C05479=1171.912,88.058,-51.231,-179.130,6.211,148.864
C05480=1171.917,87.808,-51.214,-179.132,6.209,148.865
C05481=1171.922,87.559,-51.196,-179.135,6.209,148.865
C05482=1171.927,87.310,-51.178,-179.138,6.207,148.866
C05483=1171.932,87.061,-51.160,-179.140,6.206,148.866
C05484=1171.937,86.811,-51.142,-179.143,6.205,148.867
C05485=1171.942,86.562,-51.124,-179.145,6.204,148.867
C05486=1171.946,86.312,-51.108,-179.148,6.202,148.868
C05487=1171.951,86.063,-51.090,-179.150,6.202,148.868
C05488=1171.956,85.814,-51.072,-179.153,6.200,148.869
C05489=1171.961,85.564,-51.054,-179.156,6.198,148.869
C05490=1171.966,85.315,-51.037,-179.159,6.198,148.870
C05491=1171.971,85.067,-51.019,-179.162,6.196,148.871
C05492=1171.976,84.817,-51.002,-179.164,6.195,148.871
C05493=1171.981,84.568,-50.984,-179.167,6.194,148.872
C05494=1171.986,84.318,-50.967,-179.169,6.193,148.872
C05495=1171.991,84.069,-50.950,-179.172,6.191,148.872
C05496=1171.996,83.819,-50.932,-179.175,6.191,148.873
C05497=1172.001,83.570,-50.914,-179.177,6.189,148.874
C05498=1172.006,83.321,-50.896,-179.180,6.189,148.874
C05499=1172.010,83.071,-50.880,-179.183,6.187,148.875
C05500=1172.015,82.822,-50.862,-179.185,6.186,148.875
C05501=1172.020,82.572,-50.844,-179.188,6.185,148.876
C05502=1172.025,82.323,-50.826,-179.190,6.184,148.876
C05503=1172.030,82.074,-50.810,-179.193,6.182,148.877
C05504=1172.035,81.825,-50.792,-179.196,6.182,148.877
C05505=1172.040,81.575,-50.775,-179.199,6.180,148.878
C05506=1172.044,81.326,-50.757,-179.201,6.179,148.878
C05507=1172.050,81.077,-50.740,-179.204,6.178,148.879
C05508=1172.055,80.827,-50.723,-179.206,6.177,148.879
C05509=1172.060,80.559,-50.704,-179.209,6.175,148.880
C05510=1172.065,80.290,-50.686,-179.212,6.174,148.880
C05511=1172.071,80.022,-50.667,-179.215,6.173,148.881
C05512=1172.076,79.754,-50.648,-179.218,6.172,148.881
C05513=1172.080,79.504,-50.631,-179.221,6.171,148.882
C05514=1172.086,79.255,-50.614,-179.223,6.170,148.883
C05515=1172.090,79.005,-50.596,-179.226,6.168,148.883
C05516=1172.095,78.756,-50.579,-179.228,6.167,148.884
C05517=1172.101,78.507,-50.562,-179.231,6.166,148.884
C05518=1172.106,78.258,-50.544,-179.234,6.165,148.885
C05519=1172.110,78.008,-50.528,-179.236,6.163,148.885
C05520=1172.115,77.758,-50.510,-179.239,6.163,148.886
C05521=1172.120,77.510,-50.493,-179.242,6.161,148.886
C05522=1172.125,77.260,-50.476,-179.244,6.161,148.887
C05523=1172.130,77.011,-50.459,-179.247,6.159,148.887
C05524=1172.135,76.762,-50.441,-179.250,6.159,148.888
C05525=1172.140,76.512,-50.424,-179.252,6.157,148.888
C05526=1172.144,76.262,-50.408,-179.255,6.156,148.889
C05527=1172.150,76.013,-50.390,-179.258,6.155,148.889
C05528=1172.154,75.765,-50.373,-179.260,6.154,148.890
C05529=1172.160,75.515,-50.356,-179.263,6.153,148.891
C05530=1172.164,75.265,-50.339,-179.265,6.152,148.891
C05531=1172.169,75.015,-50.322,-179.268,6.151,148.892
C05532=1172.174,74.766,-50.305,-179.271,6.149,148.892
C05533=1172.179,74.517,-50.288,-179.273,6.149,148.893
C05534=1172.184,74.268,-50.271,-179.276,6.147,148.893
C05535=1172.189,74.018,-50.254,-179.279,6.147,148.894
C05536=1172.193,73.769,-50.237,-179.281,6.145,148.894
C05537=1172.199,73.519,-50.220,-179.283,6.144,148.895
C05538=1172.204,73.270,-50.204,-179.287,6.143,148.895
C05539=1172.209,73.021,-50.186,-179.289,6.142,148.896
C05540=1172.213,72.771,-50.169,-179.292,6.140,148.896
C05541=1172.218,72.522,-50.152,-179.294,6.140,148.897
C05542=1172.223,72.273,-50.135,-179.297,6.139,148.898
C05543=1172.229,72.023,-50.118,-179.300,6.137,148.898
C05544=1172.233,71.774,-50.101,-179.302,6.137,148.899
C05545=1172.238,71.524,-50.085,-179.305,6.135,148.899
C05546=1172.243,71.275,-50.068,-179.308,6.135,148.900
C05547=1172.248,71.026,-50.051,-179.310,6.133,148.900
C05548=1172.253,70.776,-50.034,-179.313,6.132,148.901
C05549=1172.258,70.527,-50.018,-179.316,6.131,148.901
C05550=1172.263,70.277,-50.001,-179.318,6.130,148.902
C05551=1172.268,70.028,-49.984,-179.320,6.129,148.902
C05552=1172.272,69.778,-49.967,-179.323,6.128,148.903
C05553=1172.278,69.530,-49.949,-179.326,6.127,148.903
C05554=1172.283,69.280,-49.933,-179.329,6.125,148.904
C05555=1172.287,69.030,-49.917,-179.331,6.125,148.904
C05556=1172.293,68.781,-49.900,-179.334,6.123,148.905
C05557=1172.298,68.532,-49.883,-179.337,6.123,148.906
C05558=1172.302,68.282,-49.867,-179.339,6.122,148.906
C05559=1172.308,68.033,-49.850,-179.342,6.120,148.907
C05560=1172.312,67.784,-49.833,-179.344,6.120,148.907
C05561=1172.317,67.534,-49.816,-179.347,6.118,148.908
C05562=1172.323,67.285,-49.799,-179.349,6.117,148.908
C05563=1172.327,67.035,-49.783,-179.353,6.116,148.909
C05564=1172.332,66.786,-49.766,-179.355,6.115,148.909
C05565=1172.337,66.537,-49.749,-179.357,6.115,148.910
C05566=1172.342,66.287,-49.733,-179.360,6.113,148.910
C05567=1172.346,66.038,-49.716,-179.363,6.112,148.911
C05568=1172.352,65.789,-49.700,-179.365,6.111,148.911
C05569=1172.357,65.539,-49.683,-179.368,6.110,148.912
C05570=1172.362,65.290,-49.667,-179.370,6.109,148.913
C05571=1172.367,65.040,-49.650,-179.373,6.108,148.913
C05572=1172.371,64.791,-49.633,-179.376,6.107,148.914
C05573=1172.377,64.542,-49.616,-179.379,6.106,148.914
C05574=1172.382,64.292,-49.600,-179.381,6.105,148.915
C05575=1172.386,64.042,-49.584,-179.384,6.104,148.915
C05576=1172.391,63.793,-49.568,-179.386,6.103,148.916
C05577=1172.396,63.544,-49.550,-179.389,6.102,148.916
C05578=1172.401,63.295,-49.534,-179.392,6.101,148.917
C05579=1172.406,63.045,-49.518,-179.394,6.100,148.918
C05580=1172.411,62.796,-49.502,-179.397,6.099,148.918
C05581=1172.416,62.547,-49.485,-179.400,6.098,148.919
C05582=1172.421,62.296,-49.468,-179.402,6.097,148.919
C05583=1172.426,62.047,-49.452,-179.405,6.096,148.920
C05584=1172.431,61.798,-49.436,-179.407,6.095,148.920
C05585=1172.436,61.549,-49.419,-179.410,6.094,148.921
C05586=1172.441,61.299,-49.403,-179.413,6.093,148.921
C05587=1172.446,61.050,-49.387,-179.415,6.092,148.922
C05588=1172.450,60.801,-49.370,-179.417,6.091,148.922
C05589=1172.456,60.550,-49.354,-179.421,6.090,148.923
C05590=1172.461,60.302,-49.337,-179.423,6.089,148.924
C05591=1172.465,60.052,-49.321,-179.426,6.088,148.924
C05592=1172.471,59.803,-49.305,-179.428,6.087,148.925
C05593=1172.475,59.553,-49.289,-179.431,6.086,148.925
C05594=1172.481,59.304,-49.273,-179.434,6.085,148.926
C05595=1172.485,59.054,-49.256,-179.436,6.084,148.926
C05596=1172.490,58.805,-49.240,-179.438,6.083,148.927
C05597=1172.495,58.555,-49.224,-179.442,6.082,148.927
C05598=1172.501,58.306,-49.207,-179.444,6.081,148.928
C05599=1172.506,58.056,-49.191,-179.447,6.080,148.929
C05600=1172.511,57.807,-49.175,-179.449,6.079,148.929
C05601=1172.515,57.558,-49.158,-179.452,6.078,148.930
C05602=1172.521,57.308,-49.143,-179.454,6.077,148.930
C05603=1172.525,57.059,-49.126,-179.457,6.076,148.931
C05604=1172.530,56.810,-49.110,-179.459,6.075,148.931
C05605=1172.535,56.560,-49.094,-179.462,6.074,148.932
C05606=1172.540,56.311,-49.078,-179.465,6.073,148.932
C05607=1172.545,56.061,-49.061,-179.467,6.073,148.933
C05608=1172.550,55.812,-49.046,-179.470,6.071,148.934
C05609=1172.555,55.563,-49.030,-179.473,6.070,148.934
C05610=1172.560,55.313,-49.014,-179.475,6.070,148.935
C05611=1172.565,55.064,-48.998,-179.478,6.068,148.935
C05612=1172.570,54.814,-48.981,-179.481,6.068,148.936
C05613=1172.575,54.546,-48.964,-179.483,6.066,148.936
C05614=1172.581,54.277,-48.947,-179.486,6.065,148.937
C05615=1172.586,54.008,-48.930,-179.489,6.064,148.938
C05616=1172.591,53.740,-48.912,-179.492,6.064,148.938
C05617=1172.597,53.491,-48.897,-179.494,6.063,148.939
C05618=1172.601,53.241,-48.881,-179.497,6.061,148.939
C05619=1172.606,52.992,-48.864,-179.499,6.061,148.940
C05620=1172.612,52.742,-48.849,-179.502,6.060,148.941
C05621=1172.616,52.493,-48.832,-179.505,6.058,148.941
C05622=1172.622,52.243,-48.816,-179.507,6.058,148.942
C05623=1172.626,51.993,-48.800,-179.510,6.057,148.942
C05624=1172.632,51.745,-48.784,-179.513,6.056,148.943
C05625=1172.637,51.495,-48.769,-179.515,6.055,148.943
C05626=1172.641,51.245,-48.753,-179.518,6.054,148.944
C05627=1172.646,50.997,-48.737,-179.520,6.053,148.944
C05628=1172.651,50.747,-48.721,-179.523,6.052,148.945
C05629=1172.656,50.497,-48.705,-179.526,6.052,148.946
C05630=1172.662,50.248,-48.690,-179.528,6.050,148.946
C05631=1172.666,49.998,-48.673,-179.531,6.049,148.947
C05632=1172.672,49.749,-48.658,-179.533,6.049,148.947
C05633=1172.677,49.499,-48.642,-179.536,6.047,148.948
C05634=1172.681,49.250,-48.627,-179.538,6.046,148.948
C05635=1172.686,49.001,-48.610,-179.541,6.046,148.949
C05636=1172.691,48.751,-48.594,-179.544,6.044,148.949
C05637=1172.696,48.501,-48.579,-179.547,6.044,148.950
C05638=1172.702,48.252,-48.563,-179.549,6.043,148.950
C05639=1172.705,48.003,-48.547,-179.551,6.042,148.951
C05640=1172.711,47.753,-48.532,-179.555,6.041,148.952
C05641=1172.716,47.504,-48.516,-179.557,6.040,148.952
C05642=1172.721,47.255,-48.500,-179.559,6.040,148.953
C05643=1172.726,47.004,-48.484,-179.562,6.038,148.953
C05644=1172.731,46.755,-48.469,-179.565,6.038,148.954
C05645=1172.736,46.507,-48.453,-179.567,6.037,148.954
C05646=1172.741,46.256,-48.437,-179.569,6.036,148.955
C05647=1172.746,46.007,-48.422,-179.572,6.034,148.956
C05648=1172.752,45.758,-48.406,-179.575,6.034,148.956
C05649=1172.756,45.508,-48.391,-179.578,6.033,148.957
C05650=1172.761,45.258,-48.375,-179.580,6.032,148.957
C05651=1172.766,45.009,-48.359,-179.583,6.031,148.958
C05652=1172.771,44.760,-48.344,-179.585,6.030,148.959
C05653=1172.776,44.510,-48.328,-179.588,6.030,148.959
C05654=1172.781,44.260,-48.313,-179.590,6.028,148.960
C05655=1172.787,44.011,-48.297,-179.593,6.028,148.960
C05656=1172.791,43.761,-48.282,-179.595,6.027,148.961
C05657=1172.796,43.513,-48.266,-179.598,6.026,148.961
C05658=1172.801,43.263,-48.250,-179.601,6.025,148.962
C05659=1172.806,43.014,-48.235,-179.603,6.024,148.963
C05660=1172.811,42.765,-48.219,-179.606,6.024,148.963
C05661=1172.816,42.515,-48.204,-179.609,6.022,148.964
C05662=1172.821,42.265,-48.189,-179.611,6.022,148.964
C05663=1172.826,42.016,-48.173,-179.613,6.021,148.965
C05664=1172.832,41.766,-48.158,-179.616,6.020,148.965
C05665=1172.836,41.516,-48.143,-179.619,6.019,148.966
C05666=1172.841,41.267,-48.127,-179.621,6.018,148.967
C05667=1172.846,41.017,-48.112,-179.624,6.018,148.967
C05668=1172.851,40.768,-48.097,-179.626,6.017,148.968
C05669=1172.857,40.519,-48.081,-179.629,6.015,148.968
C05670=1172.861,40.269,-48.065,-179.632,6.014,148.969
C05671=1172.866,40.020,-48.050,-179.634,6.014,148.969
C05672=1172.871,39.770,-48.034,-179.637,6.014,148.970
C05673=1172.876,39.521,-48.019,-179.640,6.012,148.971
C05674=1172.881,39.272,-48.004,-179.642,6.011,148.971
C05675=1172.886,39.022,-47.988,-179.644,6.010,148.972
C05676=1172.891,38.772,-47.974,-179.647,6.010,148.972
C05677=1172.897,38.523,-47.958,-179.650,6.008,148.973
C05678=1172.901,38.274,-47.943,-179.653,6.008,148.973
C05679=1172.907,38.024,-47.927,-179.655,6.007,148.974
C05680=1172.911,37.775,-47.912,-179.657,6.006,148.975
C05681=1172.916,37.525,-47.896,-179.661,6.005,148.975
C05682=1172.922,37.275,-47.882,-179.663,6.004,148.976
C05683=1172.926,37.026,-47.867,-179.665,6.004,148.976
C05684=1172.932,36.776,-47.851,-179.668,6.003,148.977
C05685=1172.936,36.527,-47.836,-179.670,6.002,148.978
C05686=1172.942,36.278,-47.820,-179.673,6.001,148.978
C05687=1172.947,36.028,-47.806,-179.676,6.000,148.979
C05688=1172.952,35.779,-47.791,-179.678,6.000,148.979
C05689=1172.956,35.529,-47.775,-179.680,5.999,148.980
C05690=1172.962,35.280,-47.760,-179.684,5.998,148.980
C05691=1172.966,35.030,-47.745,-179.686,5.997,148.981
C05692=1172.972,34.780,-47.730,-179.688,5.996,148.982
C05693=1172.977,34.531,-47.715,-179.691,5.996,148.982
C05694=1172.982,34.281,-47.700,-179.693,5.995,148.983
C05695=1172.987,34.032,-47.685,-179.696,5.994,148.983
C05696=1172.992,33.783,-47.669,-179.699,5.993,148.984
C05697=1172.997,33.533,-47.655,-179.701,5.992,148.984
C05698=1173.001,33.283,-47.640,-179.704,5.992,148.985
C05699=1173.007,33.034,-47.624,-179.707,5.990,148.986
C05700=1173.012,32.784,-47.610,-179.709,5.990,148.986
C05701=1173.017,32.535,-47.594,-179.711,5.989,148.987
C05702=1173.022,32.286,-47.579,-179.714,5.988,148.987
C05703=1173.027,32.036,-47.564,-179.717,5.988,148.988
C05704=1173.032,31.787,-47.549,-179.719,5.986,148.989
C05705=1173.037,31.537,-47.535,-179.722,5.986,148.989
C05706=1173.042,31.288,-47.520,-179.724,5.985,148.990
C05707=1173.047,31.038,-47.505,-179.727,5.984,148.990
C05708=1173.053,30.788,-47.490,-179.730,5.984,148.991
C05709=1173.057,30.539,-47.475,-179.732,5.982,148.991
C05710=1173.062,30.290,-47.460,-179.735,5.982,148.992
C05711=1173.068,30.040,-47.445,-179.737,5.981,148.993
C05712=1173.073,29.791,-47.431,-179.740,5.980,148.993
C05713=1173.077,29.541,-47.416,-179.742,5.980,148.994
C05714=1173.083,29.292,-47.400,-179.745,5.979,148.994
C05715=1173.088,29.042,-47.386,-179.748,5.978,148.995
C05716=1173.092,28.793,-47.371,-179.750,5.977,148.996
C05717=1173.098,28.524,-47.354,-179.753,5.976,148.996
C05718=1173.103,28.255,-47.339,-179.756,5.975,148.997
C05719=1173.109,27.986,-47.322,-179.758,5.975,148.998
C05720=1173.114,27.717,-47.307,-179.761,5.974,148.998
C05721=1173.119,27.468,-47.292,-179.763,5.973,148.999
C05722=1173.125,27.218,-47.277,-179.767,5.972,148.999
C05723=1173.130,26.969,-47.263,-179.769,5.971,149.000
C05724=1173.134,26.720,-47.248,-179.771,5.971,149.001
C05725=1173.139,26.470,-47.233,-179.774,5.970,149.001
C05726=1173.145,26.220,-47.218,-179.776,5.969,149.002
C05727=1173.149,25.971,-47.203,-179.779,5.969,149.002
C05728=1173.154,25.721,-47.189,-179.782,5.967,149.003
C05729=1173.159,25.472,-47.174,-179.784,5.967,149.003
C05730=1173.165,25.222,-47.159,-179.787,5.966,149.004
C05731=1173.170,24.972,-47.145,-179.789,5.965,149.005
C05732=1173.174,24.723,-47.130,-179.792,5.965,149.005
C05733=1173.179,24.473,-47.116,-179.794,5.964,149.006
C05734=1173.185,24.223,-47.101,-179.797,5.963,149.006
C05735=1173.190,23.974,-47.086,-179.800,5.962,149.007
C05736=1173.195,23.725,-47.072,-179.802,5.961,149.008
C05737=1173.200,23.476,-47.058,-179.804,5.961,149.008
C05738=1173.205,23.226,-47.043,-179.807,5.960,149.009
C05739=1173.211,22.976,-47.028,-179.809,5.960,149.009
C05740=1173.215,22.727,-47.013,-179.812,5.959,149.010
C05741=1173.220,22.478,-46.999,-179.815,5.957,149.010
C05742=1173.225,22.228,-46.984,-179.817,5.957,149.011
C05743=1173.230,21.978,-46.970,-179.820,5.956,149.012
C05744=1173.235,21.728,-46.956,-179.822,5.956,149.012
C05745=1173.240,21.479,-46.940,-179.825,5.955,149.013
C05746=1173.245,21.229,-46.926,-179.827,5.954,149.013
C05747=1173.251,20.980,-46.912,-179.830,5.954,149.014
C05748=1173.256,20.731,-46.898,-179.833,5.953,149.015
C05749=1173.260,20.482,-46.883,-179.835,5.952,149.015
C05750=1173.265,20.232,-46.868,-179.838,5.951,149.016
C05751=1173.270,19.982,-46.854,-179.840,5.950,149.016
C05752=1173.276,19.732,-46.839,-179.842,5.950,149.017
C05753=1173.281,19.482,-46.825,-179.845,5.949,149.018
C05754=1173.286,19.233,-46.811,-179.847,5.949,149.018
C05755=1173.291,18.984,-46.796,-179.851,5.947,149.019
C05756=1173.296,18.735,-46.782,-179.853,5.946,149.019
C05757=1173.301,18.485,-46.767,-179.855,5.946,149.020
C05758=1173.306,18.235,-46.753,-179.858,5.945,149.021
C05759=1173.311,17.985,-46.739,-179.860,5.945,149.021
C05760=1173.316,17.736,-46.725,-179.863,5.944,149.022
C05761=1173.322,17.487,-46.711,-179.865,5.944,149.023
C05762=1173.326,17.238,-46.696,-179.868,5.943,149.023
C05763=1173.331,16.988,-46.681,-179.870,5.942,149.024
C05764=1173.336,16.738,-46.667,-179.873,5.941,149.024
C05765=1173.341,16.489,-46.653,-179.876,5.940,149.025
C05766=1173.347,16.240,-46.639,-179.878,5.940,149.025
C05767=1173.352,15.990,-46.625,-179.880,5.939,149.026
C05768=1173.357,15.740,-46.610,-179.883,5.938,149.027
C05769=1173.361,15.490,-46.596,-179.886,5.938,149.027
C05770=1173.366,15.241,-46.582,-179.888,5.937,149.028
C05771=1173.372,14.992,-46.568,-179.891,5.937,149.028
C05772=1173.377,14.742,-46.554,-179.893,5.936,149.029
C05773=1173.382,14.492,-46.539,-179.896,5.934,149.030
C05774=1173.387,14.243,-46.525,-179.899,5.934,149.030
C05775=1173.392,13.993,-46.511,-179.901,5.933,149.031
C05776=1173.397,13.744,-46.497,-179.903,5.933,149.031
C05777=1173.402,13.494,-46.483,-179.906,5.932,149.032
C05778=1173.407,13.244,-46.468,-179.908,5.931,149.033
C05779=1173.412,12.995,-46.454,-179.911,5.931,149.033
C05780=1173.418,12.746,-46.440,-179.913,5.930,149.034
C05781=1173.423,12.496,-46.426,-179.916,5.930,149.034
C05782=1173.428,12.246,-46.412,-179.918,5.929,149.035
C05783=1173.433,11.997,-46.397,-179.921,5.928,149.035
C05784=1173.438,11.748,-46.383,-179.924,5.927,149.036
C05785=1173.443,11.498,-46.369,-179.926,5.927,149.037
C05786=1173.448,11.247,-46.356,-179.929,5.926,149.037
C05787=1173.453,10.998,-46.341,-179.931,5.925,149.038
C05788=1173.458,10.749,-46.328,-179.933,5.924,149.038
C05789=1173.463,10.499,-46.314,-179.936,5.924,149.039
C05790=1173.468,10.250,-46.299,-179.939,5.923,149.040
C05791=1173.474,10.001,-46.286,-179.941,5.923,149.040
C05792=1173.479,9.751,-46.271,-179.944,5.922,149.041
C05793=1173.484,9.501,-46.257,-179.946,5.922,149.042
C05794=1173.489,9.252,-46.244,-179.948,5.921,149.042
C05795=1173.494,9.002,-46.230,-179.951,5.920,149.043
C05796=1173.499,8.752,-46.216,-179.954,5.920,149.043
C05797=1173.504,8.503,-46.202,-179.956,5.918,149.044
C05798=1173.509,8.254,-46.188,-179.959,5.918,149.045
C05799=1173.514,8.003,-46.174,-179.961,5.917,149.045
C05800=1173.519,7.754,-46.160,-179.964,5.916,149.046
C05801=1173.525,7.505,-46.146,-179.967,5.916,149.046
C05802=1173.529,7.255,-46.132,-179.969,5.915,149.047
C05803=1173.534,7.005,-46.119,-179.971,5.915,149.048
C05804=1173.540,6.756,-46.105,-179.974,5.914,149.048
C05805=1173.545,6.506,-46.090,-179.976,5.913,149.049
C05806=1173.550,6.257,-46.076,-179.979,5.913,149.049
C05807=1173.555,6.007,-46.064,-179.982,5.912,149.050
C05808=1173.560,5.758,-46.049,-179.984,5.912,149.051
C05809=1173.565,5.509,-46.035,-179.986,5.911,149.051
C05810=1173.570,5.259,-46.021,-179.989,5.910,149.052
C05811=1173.575,5.009,-46.008,-179.991,5.910,149.052
C05812=1173.581,4.760,-45.994,-179.994,5.909,149.053
C05813=1173.585,4.510,-45.980,-179.996,5.908,149.054
C05814=1173.591,4.260,-45.966,-179.999,5.908,149.054
C05815=1173.596,4.011,-45.953,179.999,5.908,149.055
C05816=1173.601,3.761,-45.939,179.996,5.906,149.055
C05817=1173.606,3.512,-45.926,179.993,5.905,149.056
C05818=1173.611,3.262,-45.912,179.991,5.905,149.057
C05819=1173.616,3.012,-45.898,179.988,5.904,149.057
C05820=1173.621,2.763,-45.884,179.986,5.904,149.058
C05821=1173.627,2.494,-45.869,179.983,5.903,149.059
C05822=1173.632,2.224,-45.854,179.981,5.903,149.059
C05823=1173.637,1.955,-45.840,179.978,5.902,149.060
C05824=1173.643,1.686,-45.825,179.976,5.901,149.060
C05825=1173.648,1.436,-45.812,179.973,5.901,149.061
C05826=1173.654,1.187,-45.798,179.970,5.899,149.062
C05827=1173.658,0.937,-45.785,179.968,5.899,149.062
C05828=1173.663,0.687,-45.771,179.965,5.898,149.063
C05829=1173.669,0.438,-45.758,179.963,5.898,149.063
C05830=1173.673,0.188,-45.744,179.960,5.897,149.064
C05831=1173.679,-0.061,-45.731,179.957,5.897,149.065
C05832=1173.683,-0.311,-45.717,179.955,5.896,149.065
C05833=1173.689,-0.560,-45.704,179.953,5.895,149.066
C05834=1173.694,-0.810,-45.690,179.950,5.895,149.067
C05835=1173.699,-1.059,-45.677,179.948,5.894,149.067
C05836=1173.704,-1.309,-45.663,179.945,5.894,149.068
C05837=1173.710,-1.559,-45.649,179.943,5.893,149.069
C05838=1173.714,-1.808,-45.636,179.940,5.892,149.069
C05839=1173.720,-2.058,-45.623,179.938,5.892,149.070
C05840=1173.724,-2.307,-45.609,179.936,5.891,149.070
C05841=1173.730,-2.557,-45.596,179.933,5.891,149.071
C05842=1173.735,-2.807,-45.581,179.930,5.890,149.071
C05843=1173.740,-3.056,-45.569,179.928,5.889,149.072
C05844=1173.746,-3.306,-45.555,179.925,5.889,149.073
C05845=1173.751,-3.555,-45.542,179.923,5.888,149.073
C05846=1173.756,-3.805,-45.528,179.921,5.887,149.074
C05847=1173.761,-4.054,-45.515,179.918,5.887,149.074
C05848=1173.766,-4.304,-45.501,179.915,5.887,149.075
C05849=1173.771,-4.554,-45.489,179.913,5.886,149.076
C05850=1173.776,-4.803,-45.475,179.910,5.885,149.076
C05851=1173.781,-5.053,-45.462,179.908,5.885,149.077
C05852=1173.786,-5.303,-45.448,179.906,5.884,149.077
C05853=1173.791,-5.552,-45.435,179.903,5.884,149.078
C05854=1173.796,-5.802,-45.422,179.900,5.883,149.079
C05855=1173.802,-6.051,-45.409,179.898,5.882,149.079
C05856=1173.806,-6.301,-45.395,179.895,5.882,149.080
C05857=1173.812,-6.550,-45.382,179.893,5.881,149.080
C05858=1173.817,-6.801,-45.369,179.891,5.880,149.081
C05859=1173.822,-7.049,-45.355,179.888,5.880,149.082
C05860=1173.828,-7.299,-45.342,179.886,5.879,149.082
C05861=1173.832,-7.549,-45.329,179.883,5.879,149.083
C05862=1173.838,-7.799,-45.316,179.880,5.878,149.084
C05863=1173.842,-8.048,-45.302,179.878,5.877,149.084
C05864=1173.848,-8.298,-45.289,179.876,5.877,149.085
C05865=1173.853,-8.548,-45.276,179.873,5.877,149.086
C05866=1173.858,-8.797,-45.263,179.871,5.876,149.086
C05867=1173.863,-9.046,-45.250,179.869,5.876,149.087
C05868=1173.868,-9.296,-45.237,179.866,5.876,149.087
C05869=1173.874,-9.546,-45.223,179.864,5.875,149.088
C05870=1173.878,-9.796,-45.210,179.861,5.874,149.089
C05871=1173.884,-10.045,-45.197,179.859,5.874,149.089
C05872=1173.889,-10.294,-45.184,179.856,5.873,149.090
C05873=1173.893,-10.544,-45.171,179.854,5.873,149.090
C05874=1173.899,-10.794,-45.158,179.852,5.872,149.091
C05875=1173.904,-11.044,-45.145,179.849,5.871,149.092
C05876=1173.909,-11.293,-45.132,179.846,5.871,149.092
C05877=1173.915,-11.543,-45.119,179.844,5.870,149.093
C05878=1173.919,-11.792,-45.105,179.841,5.870,149.093
C05879=1173.925,-12.042,-45.092,179.839,5.869,149.094
C05880=1173.930,-12.291,-45.079,179.837,5.868,149.095
C05881=1173.934,-12.541,-45.066,179.834,5.868,149.095
C05882=1173.940,-12.791,-45.053,179.831,5.867,149.096
C05883=1173.945,-13.041,-45.040,179.829,5.867,149.096
C05884=1173.950,-13.290,-45.028,179.826,5.866,149.097
C05885=1173.956,-13.540,-45.015,179.824,5.866,149.098
C05886=1173.960,-13.790,-45.002,179.822,5.865,149.098
C05887=1173.965,-14.039,-44.989,179.819,5.864,149.099
C05888=1173.971,-14.288,-44.976,179.816,5.864,149.100
C05889=1173.976,-14.539,-44.963,179.814,5.863,149.100
C05890=1173.981,-14.787,-44.949,179.812,5.863,149.101
C05891=1173.986,-15.037,-44.937,179.810,5.863,149.101
C05892=1173.991,-15.287,-44.923,179.807,5.862,149.102
C05893=1173.996,-15.536,-44.911,179.805,5.862,149.103
C05894=1174.001,-15.786,-44.898,179.802,5.861,149.103
C05895=1174.006,-16.035,-44.886,179.800,5.860,149.104
C05896=1174.012,-16.285,-44.872,179.797,5.860,149.105
C05897=1174.017,-16.535,-44.859,179.795,5.859,149.105
C05898=1174.022,-16.784,-44.847,179.792,5.859,149.106
C05899=1174.027,-17.035,-44.834,179.790,5.858,149.106
C05900=1174.033,-17.284,-44.821,179.787,5.857,149.107
C05901=1174.038,-17.533,-44.809,179.785,5.857,149.108
C05902=1174.043,-17.783,-44.796,179.782,5.857,149.108
C05903=1174.047,-18.033,-44.783,179.780,5.856,149.109
C05904=1174.053,-18.282,-44.770,179.777,5.855,149.109
C05905=1174.058,-18.532,-44.757,179.775,5.856,149.110
C05906=1174.063,-18.782,-44.744,179.773,5.855,149.111
C05907=1174.068,-19.031,-44.732,179.770,5.854,149.111
C05908=1174.073,-19.280,-44.719,179.768,5.854,149.112
C05909=1174.079,-19.530,-44.706,179.766,5.853,149.112
C05910=1174.083,-19.780,-44.693,179.763,5.853,149.113
C05911=1174.089,-20.030,-44.681,179.761,5.852,149.114
C05912=1174.094,-20.279,-44.669,179.758,5.851,149.114
C05913=1174.099,-20.529,-44.656,179.755,5.851,149.115
C05914=1174.105,-20.778,-44.643,179.753,5.850,149.115
C05915=1174.110,-21.028,-44.630,179.751,5.850,149.116
C05916=1174.115,-21.278,-44.617,179.748,5.850,149.117
C05917=1174.120,-21.527,-44.605,179.746,5.849,149.117
C05918=1174.125,-21.777,-44.593,179.744,5.849,149.118
C05919=1174.130,-22.027,-44.580,179.741,5.848,149.119
C05920=1174.135,-22.276,-44.567,179.739,5.847,149.119
C05921=1174.141,-22.526,-44.554,179.736,5.847,149.120
C05922=1174.146,-22.776,-44.542,179.733,5.847,149.121
C05923=1174.151,-23.025,-44.529,179.731,5.846,149.121
C05924=1174.156,-23.275,-44.516,179.729,5.845,149.122
C05925=1174.161,-23.544,-44.503,179.726,5.845,149.122
C05926=1174.167,-23.815,-44.490,179.723,5.844,149.123
C05927=1174.173,-24.084,-44.476,179.721,5.844,149.124
C05928=1174.178,-24.353,-44.463,179.718,5.843,149.124
C05929=1174.183,-24.603,-44.450,179.716,5.843,149.125
C05930=1174.189,-24.853,-44.438,179.713,5.842,149.126
C05931=1174.194,-25.103,-44.425,179.711,5.841,149.126
C05932=1174.199,-25.352,-44.412,179.709,5.842,149.127
C05933=1174.204,-25.602,-44.400,179.706,5.841,149.128
C05934=1174.210,-25.852,-44.387,179.704,5.841,149.128
C05935=1174.215,-26.101,-44.375,179.701,5.840,149.129
C05936=1174.220,-26.351,-44.363,179.699,5.840,149.129
C05937=1174.225,-26.601,-44.350,179.697,5.839,149.130
C05938=1174.230,-26.850,-44.337,179.694,5.838,149.131
C05939=1174.235,-27.100,-44.326,179.692,5.838,149.131
C05940=1174.240,-27.349,-44.313,179.689,5.837,149.132
C05941=1174.245,-27.599,-44.300,179.687,5.837,149.132
C05942=1174.251,-27.849,-44.288,179.685,5.837,149.133
C05943=1174.256,-28.098,-44.276,179.682,5.836,149.134
C05944=1174.261,-28.349,-44.264,179.679,5.836,149.134
C05945=1174.266,-28.598,-44.251,179.677,5.835,149.135
C05946=1174.271,-28.847,-44.238,179.675,5.835,149.135
C05947=1174.276,-29.097,-44.227,179.672,5.834,149.136
C05948=1174.282,-29.347,-44.214,179.670,5.833,149.137
C05949=1174.287,-29.597,-44.202,179.668,5.834,149.137
C05950=1174.292,-29.846,-44.189,179.665,5.833,149.138
C05951=1174.297,-30.095,-44.177,179.663,5.832,149.139
C05952=1174.303,-30.345,-44.165,179.660,5.832,149.139
C05953=1174.307,-30.594,-44.153,179.658,5.831,149.140
C05954=1174.312,-30.845,-44.141,179.655,5.831,149.140
C05955=1174.317,-31.094,-44.128,179.653,5.830,149.141
C05956=1174.322,-31.344,-44.116,179.651,5.830,149.142
C05957=1174.328,-31.593,-44.104,179.648,5.830,149.142
C05958=1174.333,-31.843,-44.092,179.646,5.829,149.143
C05959=1174.338,-32.093,-44.079,179.644,5.829,149.143
C05960=1174.344,-32.342,-44.067,179.641,5.828,149.144
C05961=1174.349,-32.592,-44.055,179.638,5.828,149.145
C05962=1174.354,-32.842,-44.043,179.636,5.827,149.145
C05963=1174.359,-33.091,-44.030,179.634,5.827,149.146
C05964=1174.364,-33.341,-44.019,179.631,5.827,149.147
C05965=1174.369,-33.591,-44.007,179.629,5.826,149.147
C05966=1174.375,-33.840,-43.994,179.627,5.826,149.148
C05967=1174.380,-34.090,-43.982,179.624,5.825,149.149
C05968=1174.385,-34.339,-43.970,179.622,5.824,149.149
C05969=1174.391,-34.589,-43.958,179.620,5.825,149.150
C05970=1174.396,-34.838,-43.945,179.617,5.824,149.150
C05971=1174.400,-35.088,-43.934,179.615,5.823,149.151
C05972=1174.406,-35.338,-43.922,179.612,5.823,149.152
C05973=1174.411,-35.587,-43.910,179.610,5.822,149.152
C05974=1174.416,-35.837,-43.898,179.607,5.822,149.153
C05975=1174.422,-36.087,-43.886,179.605,5.821,149.153
C05976=1174.427,-36.337,-43.873,179.603,5.821,149.154
C05977=1174.432,-36.586,-43.862,179.600,5.821,149.155
C05978=1174.437,-36.835,-43.849,179.598,5.820,149.155
C05979=1174.442,-37.085,-43.837,179.596,5.820,149.156
C05980=1174.448,-37.335,-43.826,179.593,5.819,149.157
C05981=1174.453,-37.585,-43.813,179.590,5.819,149.157
C05982=1174.457,-37.834,-43.802,179.589,5.819,149.158
C05983=1174.463,-38.084,-43.790,179.586,5.818,149.158
C05984=1174.468,-38.334,-43.778,179.584,5.817,149.159
C05985=1174.473,-38.583,-43.765,179.581,5.817,149.160
C05986=1174.479,-38.833,-43.753,179.578,5.817,149.160
C05987=1174.483,-39.083,-43.742,179.577,5.817,149.161
C05988=1174.489,-39.332,-43.730,179.574,5.816,149.161
C05989=1174.494,-39.582,-43.718,179.572,5.816,149.162
C05990=1174.499,-39.832,-43.706,179.569,5.815,149.163
C05991=1174.504,-40.082,-43.694,179.567,5.814,149.163
C05992=1174.509,-40.331,-43.682,179.564,5.814,149.164
C05993=1174.515,-40.581,-43.670,179.562,5.814,149.164
C05994=1174.519,-40.831,-43.659,179.560,5.814,149.165
C05995=1174.525,-41.081,-43.647,179.558,5.813,149.166
C05996=1174.530,-41.331,-43.635,179.555,5.812,149.166
C05997=1174.536,-41.579,-43.623,179.552,5.812,149.167
C05998=1174.541,-41.829,-43.611,179.551,5.812,149.168
C05999=1174.546,-42.079,-43.600,179.548,5.811,149.168
C06000=1174.552,-42.329,-43.588,179.545,5.811,149.169
C06001=1174.556,-42.578,-43.576,179.543,5.810,149.169
C06002=1174.561,-42.828,-43.564,179.540,5.810,149.170
C06003=1174.567,-43.078,-43.552,179.538,5.810,149.171
C06004=1174.571,-43.327,-43.541,179.536,5.809,149.171
C06005=1174.577,-43.577,-43.529,179.534,5.809,149.172
C06006=1174.582,-43.827,-43.517,179.531,5.808,149.172
C06007=1174.587,-44.077,-43.506,179.529,5.808,149.173
C06008=1174.593,-44.326,-43.494,179.527,5.808,149.174
C06009=1174.598,-44.576,-43.482,179.524,5.807,149.174
C06010=1174.603,-44.825,-43.470,179.522,5.807,149.175
C06011=1174.608,-45.075,-43.458,179.519,5.806,149.176
C06012=1174.613,-45.324,-43.447,179.517,5.806,149.176
C06013=1174.618,-45.574,-43.435,179.515,5.806,149.177
C06014=1174.624,-45.824,-43.423,179.513,5.805,149.177
C06015=1174.629,-46.073,-43.412,179.510,5.805,149.178
C06016=1174.635,-46.323,-43.400,179.507,5.804,149.179
C06017=1174.639,-46.573,-43.389,179.505,5.803,149.179
C06018=1174.645,-46.823,-43.377,179.503,5.804,149.180
C06019=1174.650,-47.073,-43.365,179.500,5.803,149.181
C06020=1174.655,-47.322,-43.354,179.498,5.803,149.181
C06021=1174.660,-47.572,-43.342,179.496,5.802,149.182
C06022=1174.666,-47.821,-43.331,179.494,5.803,149.183
C06023=1174.671,-48.071,-43.319,179.491,5.802,149.183
C06024=1174.676,-48.321,-43.308,179.489,5.801,149.184
C06025=1174.681,-48.571,-43.296,179.486,5.801,149.184
C06026=1174.686,-48.821,-43.284,179.484,5.800,149.185
C06027=1174.692,-49.070,-43.273,179.482,5.800,149.186
C06028=1174.697,-49.319,-43.261,179.480,5.800,149.186
C06029=1174.703,-49.590,-43.248,179.477,5.799,149.187
C06030=1174.708,-49.861,-43.236,179.474,5.799,149.187
C06031=1174.713,-50.130,-43.224,179.472,5.798,149.188
C06032=1174.719,-50.401,-43.212,179.469,5.798,149.189
C06033=1174.724,-50.651,-43.200,179.467,5.797,149.189
C06034=1174.730,-50.900,-43.189,179.465,5.798,149.190
C06035=1174.735,-51.150,-43.177,179.462,5.797,149.191
C06036=1174.740,-51.400,-43.166,179.460,5.796,149.191
C06037=1174.745,-51.649,-43.154,179.457,5.796,149.192
C06038=1174.750,-51.899,-43.143,179.456,5.796,149.192
C06039=1174.756,-52.149,-43.132,179.453,5.795,149.193
C06040=1174.761,-52.399,-43.121,179.450,5.795,149.194
C06041=1174.766,-52.649,-43.109,179.448,5.794,149.194
C06042=1174.771,-52.898,-43.098,179.446,5.795,149.195
C06043=1174.777,-53.147,-43.086,179.444,5.794,149.195
C06044=1174.782,-53.397,-43.075,179.441,5.793,149.196
C06045=1174.787,-53.647,-43.063,179.438,5.793,149.197
C06046=1174.792,-53.897,-43.052,179.437,5.793,149.197
C06047=1174.797,-54.146,-43.041,179.434,5.793,149.198
C06048=1174.803,-54.396,-43.029,179.431,5.792,149.199
C06049=1174.808,-54.646,-43.018,179.429,5.791,149.199
C06050=1174.813,-54.896,-43.006,179.427,5.792,149.200
C06051=1174.818,-55.145,-42.995,179.425,5.791,149.200
C06052=1174.823,-55.395,-42.985,179.422,5.790,149.201
C06053=1174.829,-55.645,-42.973,179.420,5.790,149.202
C06054=1174.833,-55.894,-42.962,179.418,5.790,149.202
C06055=1174.839,-56.144,-42.950,179.415,5.790,149.203
C06056=1174.844,-56.394,-42.940,179.413,5.789,149.204
C06057=1174.849,-56.643,-42.928,179.411,5.788,149.204
C06058=1174.855,-56.893,-42.917,179.409,5.789,149.205
C06059=1174.860,-57.142,-42.905,179.406,5.788,149.205
C06060=1174.865,-57.393,-42.895,179.404,5.788,149.206
C06061=1174.871,-57.642,-42.883,179.401,5.787,149.207
C06062=1174.876,-57.891,-42.872,179.399,5.787,149.207
C06063=1174.880,-58.141,-42.861,179.397,5.787,149.208
C06064=1174.886,-58.392,-42.850,179.395,5.786,149.208
C06065=1174.891,-58.641,-42.839,179.392,5.786,149.209
C06066=1174.896,-58.890,-42.827,179.390,5.786,149.210
C06067=1174.902,-59.141,-42.816,179.388,5.785,149.210
C06068=1174.907,-59.390,-42.805,179.385,5.785,149.211
C06069=1174.912,-59.639,-42.794,179.383,5.785,149.212
C06070=1174.917,-59.890,-42.783,179.381,5.784,149.212
C06071=1174.923,-60.139,-42.772,179.378,5.784,149.213
C06072=1174.927,-60.388,-42.761,179.376,5.783,149.213
C06073=1174.933,-60.639,-42.749,179.374,5.783,149.214
C06074=1174.938,-60.888,-42.738,179.372,5.783,149.215
C06075=1174.943,-61.138,-42.728,179.369,5.782,149.215
C06076=1174.948,-61.388,-42.717,179.366,5.782,149.216
C06077=1174.954,-61.637,-42.705,179.365,5.782,149.216
C06078=1174.959,-61.887,-42.695,179.362,5.781,149.217
C06079=1174.964,-62.136,-42.684,179.360,5.781,149.218
C06080=1174.969,-62.386,-42.673,179.358,5.781,149.218
C06081=1174.975,-62.636,-42.661,179.355,5.781,149.219
C06082=1174.980,-62.885,-42.650,179.353,5.780,149.220
C06083=1174.985,-63.135,-42.640,179.350,5.779,149.220
C06084=1174.990,-63.385,-42.628,179.349,5.779,149.221
C06085=1174.996,-63.635,-42.618,179.346,5.779,149.221
C06086=1175.001,-63.885,-42.606,179.343,5.779,149.222
C06087=1175.007,-64.134,-42.596,179.342,5.779,149.223
C06088=1175.011,-64.384,-42.585,179.339,5.778,149.223
C06089=1175.016,-64.634,-42.574,179.337,5.777,149.224
C06090=1175.022,-64.883,-42.563,179.334,5.777,149.225
C06091=1175.027,-65.133,-42.552,179.332,5.777,149.225
C06092=1175.033,-65.382,-42.541,179.330,5.776,149.226
C06093=1175.038,-65.633,-42.531,179.327,5.776,149.226
C06094=1175.042,-65.882,-42.519,179.326,5.776,149.227
C06095=1175.049,-66.132,-42.509,179.323,5.776,149.228
C06096=1175.053,-66.382,-42.497,179.320,5.775,149.228
C06097=1175.059,-66.631,-42.487,179.319,5.775,149.229
C06098=1175.064,-66.881,-42.476,179.316,5.775,149.230
C06099=1175.069,-67.130,-42.466,179.314,5.774,149.230
C06100=1175.074,-67.380,-42.454,179.311,5.774,149.231
C06101=1175.080,-67.630,-42.443,179.309,5.774,149.231
C06102=1175.085,-67.880,-42.433,179.307,5.773,149.232
C06103=1175.090,-68.130,-42.422,179.304,5.773,149.233
C06104=1175.095,-68.379,-42.411,179.303,5.773,149.233
C06105=1175.100,-68.629,-42.400,179.300,5.772,149.234
C06106=1175.106,-68.879,-42.390,179.298,5.772,149.234
C06107=1175.111,-69.129,-42.379,179.296,5.772,149.235
C06108=1175.117,-69.378,-42.368,179.293,5.772,149.236
C06109=1175.122,-69.628,-42.357,179.291,5.771,149.236
C06110=1175.127,-69.877,-42.346,179.289,5.771,149.237
C06111=1175.132,-70.127,-42.336,179.287,5.770,149.237
C06112=1175.138,-70.377,-42.325,179.284,5.770,149.238
C06113=1175.142,-70.627,-42.314,179.282,5.770,149.239
C06114=1175.148,-70.876,-42.304,179.280,5.770,149.239
C06115=1175.153,-71.126,-42.293,179.277,5.769,149.240
C06116=1175.158,-71.375,-42.282,179.275,5.769,149.240
C06117=1175.163,-71.626,-42.272,179.273,5.769,149.241
C06118=1175.169,-71.875,-42.262,179.270,5.768,149.242
C06119=1175.174,-72.125,-42.250,179.268,5.768,149.242
C06120=1175.180,-72.375,-42.240,179.266,5.768,149.243
C06121=1175.185,-72.625,-42.229,179.264,5.767,149.243
C06122=1175.190,-72.874,-42.219,179.261,5.767,149.244
C06123=1175.195,-73.124,-42.208,179.259,5.767,149.245
C06124=1175.201,-73.374,-42.197,179.257,5.766,149.245
C06125=1175.206,-73.624,-42.187,179.254,5.766,149.246
C06126=1175.211,-73.873,-42.177,179.252,5.766,149.247
C06127=1175.216,-74.123,-42.165,179.250,5.766,149.247
C06128=1175.222,-74.372,-42.155,179.247,5.765,149.248
C06129=1175.227,-74.622,-42.145,179.245,5.765,149.248
C06130=1175.232,-74.872,-42.134,179.243,5.764,149.249
C06131=1175.238,-75.121,-42.123,179.241,5.764,149.250
C06132=1175.243,-75.371,-42.113,179.238,5.764,149.250
C06133=1175.249,-75.642,-42.102,179.236,5.764,149.251
C06134=1175.254,-75.914,-42.091,179.234,5.763,149.252
C06135=1175.260,-76.185,-42.078,179.231,5.763,149.252
C06136=1175.266,-76.455,-42.068,179.229,5.763,149.253
C06137=1175.271,-76.705,-42.057,179.227,5.762,149.253
C06138=1175.276,-76.955,-42.047,179.224,5.762,149.254
C06139=1175.281,-77.205,-42.036,179.222,5.762,149.255
C06140=1175.287,-77.454,-42.026,179.220,5.762,149.255
C06141=1175.292,-77.704,-42.015,179.218,5.761,149.256
C06142=1175.297,-77.954,-42.005,179.215,5.761,149.257
C06143=1175.303,-78.203,-41.995,179.213,5.761,149.257
C06144=1175.308,-78.454,-41.984,179.211,5.760,149.258
C06145=1175.313,-78.703,-41.974,179.209,5.760,149.258
C06146=1175.319,-78.953,-41.964,179.206,5.760,149.259
C06147=1175.324,-79.202,-41.952,179.204,5.759,149.260
C06148=1175.329,-79.452,-41.942,179.202,5.759,149.260
C06149=1175.333,-79.702,-41.932,179.199,5.759,149.261
C06150=1175.339,-79.951,-41.922,179.198,5.759,149.261
C06151=1175.345,-80.201,-41.912,179.195,5.758,149.262
C06152=1175.350,-80.451,-41.901,179.192,5.758,149.263
C06153=1175.355,-80.701,-41.891,179.191,5.758,149.263
C06154=1175.360,-80.951,-41.880,179.188,5.758,149.264
C06155=1175.366,-81.201,-41.870,179.186,5.757,149.264
C06156=1175.371,-81.450,-41.860,179.184,5.757,149.265
C06157=1175.376,-81.700,-41.849,179.182,5.756,149.266
C06158=1175.381,-81.950,-41.840,179.179,5.756,149.266
C06159=1175.387,-82.199,-41.829,179.177,5.756,149.267
C06160=1175.392,-82.449,-41.819,179.175,5.756,149.267
C06161=1175.398,-82.699,-41.809,179.172,5.755,149.268
C06162=1175.403,-82.948,-41.798,179.171,5.755,149.269
C06163=1175.408,-83.199,-41.788,179.168,5.755,149.269
C06164=1175.413,-83.448,-41.778,179.166,5.755,149.270
C06165=1175.419,-83.697,-41.768,179.164,5.754,149.271
C06166=1175.424,-83.948,-41.758,179.161,5.754,149.271
C06167=1175.429,-84.197,-41.747,179.159,5.754,149.272
C06168=1175.435,-84.447,-41.737,179.157,5.753,149.272
C06169=1175.439,-84.697,-41.727,179.154,5.753,149.273
C06170=1175.445,-84.946,-41.717,179.153,5.753,149.273
C06171=1175.450,-85.196,-41.707,179.150,5.752,149.274
C06172=1175.455,-85.446,-41.696,179.148,5.753,149.275
C06173=1175.461,-85.696,-41.686,179.146,5.752,149.275
C06174=1175.466,-85.945,-41.676,179.143,5.752,149.276
C06175=1175.471,-86.195,-41.666,179.142,5.752,149.277
C06176=1175.476,-86.445,-41.656,179.139,5.751,149.277
C06177=1175.482,-86.694,-41.645,179.137,5.750,149.278
C06178=1175.487,-86.944,-41.636,179.135,5.751,149.278
C06179=1175.492,-87.194,-41.626,179.133,5.750,149.279
C06180=1175.498,-87.444,-41.616,179.130,5.750,149.280
C06181=1175.503,-87.693,-41.605,179.128,5.750,149.280
C06182=1175.507,-87.943,-41.595,179.126,5.749,149.281
C06183=1175.513,-88.193,-41.585,179.124,5.749,149.281
C06184=1175.519,-88.442,-41.575,179.121,5.749,149.282
C06185=1175.525,-88.693,-41.566,179.120,5.749,149.283
C06186=1175.529,-88.942,-41.556,179.117,5.749,149.283
C06187=1175.534,-89.192,-41.545,179.114,5.748,149.284
C06188=1175.540,-89.442,-41.535,179.113,5.748,149.284
C06189=1175.545,-89.691,-41.526,179.110,5.748,149.285
C06190=1175.550,-89.941,-41.515,179.109,5.748,149.286
C06191=1175.556,-90.191,-41.505,179.106,5.747,149.286
C06192=1175.561,-90.440,-41.496,179.104,5.747,149.287
C06193=1175.566,-90.690,-41.486,179.102,5.747,149.288
C06194=1175.571,-90.940,-41.475,179.099,5.746,149.288
C06195=1175.577,-91.190,-41.466,179.097,5.747,149.289
C06196=1175.582,-91.440,-41.456,179.095,5.746,149.289
C06197=1175.588,-91.689,-41.446,179.092,5.745,149.290
C06198=1175.593,-91.939,-41.435,179.091,5.745,149.290
C06199=1175.597,-92.189,-41.426,179.088,5.745,149.291
C06200=1175.603,-92.439,-41.416,179.087,5.745,149.292
C06201=1175.608,-92.688,-41.406,179.084,5.745,149.292
C06202=1175.614,-92.938,-41.396,179.082,5.744,149.293
C06203=1175.619,-93.188,-41.386,179.080,5.744,149.293
C06204=1175.624,-93.438,-41.377,179.077,5.744,149.294
C06205=1175.630,-93.687,-41.367,179.075,5.744,149.295
C06206=1175.635,-93.937,-41.356,179.073,5.743,149.295
C06207=1175.640,-94.187,-41.347,179.070,5.743,149.296
C06208=1175.645,-94.437,-41.337,179.069,5.743,149.296
C06209=1175.650,-94.686,-41.327,179.066,5.742,149.297
C06210=1175.656,-94.936,-41.318,179.065,5.742,149.298
C06211=1175.662,-95.186,-41.308,179.062,5.742,149.298
C06212=1175.667,-95.435,-41.298,179.060,5.741,149.299
C06213=1175.672,-95.686,-41.288,179.058,5.742,149.299
C06214=1175.677,-95.935,-41.278,179.055,5.741,149.300
C06215=1175.682,-96.185,-41.268,179.053,5.741,149.301
C06216=1175.688,-96.435,-41.259,179.051,5.740,149.301
C06217=1175.693,-96.684,-41.249,179.049,5.741,149.302
C06218=1175.699,-96.934,-41.240,179.047,5.740,149.302
C06219=1175.703,-97.184,-41.230,179.044,5.740,149.303
C06220=1175.709,-97.434,-41.219,179.043,5.740,149.304
C06221=1175.714,-97.684,-41.211,179.040,5.739,149.304
C06222=1175.720,-97.933,-41.200,179.038,5.739,149.305
C06223=1175.726,-98.183,-41.191,179.036,5.739,149.305
C06224=1175.730,-98.432,-41.181,179.034,5.739,149.306
C06225=1175.736,-98.682,-41.171,179.031,5.739,149.307
C06226=1175.741,-98.932,-41.162,179.029,5.738,149.307
C06227=1175.746,-99.182,-41.152,179.027,5.738,149.308
C06228=1175.751,-99.432,-41.143,179.025,5.737,149.308
C06229=1175.757,-99.682,-41.132,179.023,5.738,149.309
C06230=1175.762,-99.931,-41.124,179.021,5.737,149.310
C06231=1175.768,-100.181,-41.113,179.019,5.737,149.310
C06232=1175.773,-100.431,-41.104,179.016,5.737,149.311
C06233=1175.778,-100.680,-41.094,179.014,5.736,149.311
C06234=1175.784,-100.930,-41.085,179.012,5.736,149.312
C06235=1175.789,-101.180,-41.075,179.009,5.736,149.313
C06236=1175.794,-101.430,-41.066,179.008,5.736,149.313
C06237=1175.800,-101.701,-41.055,179.005,5.736,149.314
C06238=1175.806,-101.973,-41.044,179.003,5.735,149.315
C06239=1175.811,-102.245,-41.034,179.001,5.735,149.315
C06240=1175.817,-102.517,-41.024,178.998,5.735,149.316
C06241=1175.823,-102.767,-41.015,178.996,5.734,149.316
C06242=1175.828,-103.016,-41.005,178.994,5.734,149.317
C06243=1175.833,-103.266,-40.996,178.992,5.734,149.317
C06244=1175.838,-103.516,-40.986,178.990,5.734,149.318
C06245=1175.843,-103.766,-40.977,178.987,5.733,149.319
C06246=1175.849,-104.015,-40.967,178.985,5.734,149.319
C06247=1175.854,-104.265,-40.958,178.983,5.733,149.320
C06248=1175.859,-104.515,-40.949,178.981,5.733,149.321
C06249=1175.865,-104.764,-40.939,178.979,5.733,149.321
C06250=1175.870,-105.014,-40.930,178.976,5.732,149.322
C06251=1175.876,-105.264,-40.920,178.975,5.732,149.322
C06252=1175.880,-105.514,-40.910,178.972,5.732,149.323
C06253=1175.886,-105.764,-40.901,178.970,5.732,149.323
C06254=1175.891,-106.014,-40.891,178.968,5.731,149.324
C06255=1175.896,-106.264,-40.882,178.966,5.731,149.325
C06256=1175.902,-106.513,-40.872,178.964,5.731,149.325
C06257=1175.907,-106.763,-40.863,178.962,5.731,149.326
C06258=1175.912,-107.013,-40.854,178.960,5.730,149.326
C06259=1175.918,-107.262,-40.844,178.957,5.730,149.327
C06260=1175.923,-107.512,-40.835,178.955,5.730,149.327
C06261=1175.928,-107.762,-40.826,178.953,5.730,149.328
C06262=1175.934,-108.012,-40.816,178.951,5.730,149.329
C06263=1175.939,-108.261,-40.807,178.948,5.729,149.329
C06264=1175.944,-108.511,-40.798,178.947,5.729,149.330
C06265=1175.950,-108.761,-40.788,178.945,5.728,149.330
C06266=1175.955,-109.011,-40.779,178.943,5.729,149.331
C06267=1175.960,-109.261,-40.770,178.940,5.728,149.332
C06268=1175.966,-109.511,-40.761,178.938,5.728,149.332
C06269=1175.971,-109.760,-40.751,178.936,5.728,149.333
C06270=1175.976,-110.010,-40.742,178.934,5.728,149.333
C06271=1175.982,-110.260,-40.733,178.932,5.727,149.334
C06272=1175.987,-110.509,-40.723,178.929,5.727,149.335
C06273=1175.992,-110.759,-40.714,178.928,5.727,149.335
C06274=1175.998,-111.009,-40.705,178.925,5.726,149.336
C06275=1176.003,-111.259,-40.696,178.923,5.727,149.336
C06276=1176.008,-111.509,-40.687,178.921,5.726,149.337
C06277=1176.013,-111.758,-40.677,178.919,5.726,149.338
C06278=1176.019,-112.008,-40.668,178.917,5.726,149.338
C06279=1176.024,-112.258,-40.659,178.915,5.726,149.339
C06280=1176.030,-112.507,-40.650,178.913,5.725,149.339
C06281=1176.035,-112.757,-40.640,178.910,5.726,149.340
C06282=1176.041,-113.007,-40.631,178.908,5.725,149.340
C06283=1176.046,-113.257,-40.622,178.907,5.725,149.341
C06284=1176.051,-113.506,-40.614,178.904,5.724,149.342
C06285=1176.057,-113.757,-40.604,178.902,5.724,149.342
C06286=1176.062,-114.006,-40.595,178.900,5.724,149.343
C06287=1176.067,-114.256,-40.586,178.898,5.724,149.343
C06288=1176.072,-114.505,-40.577,178.895,5.724,149.344
C06289=1176.078,-114.756,-40.567,178.894,5.724,149.345
C06290=1176.083,-115.006,-40.558,178.892,5.723,149.345
C06291=1176.088,-115.255,-40.549,178.890,5.723,149.346
C06292=1176.093,-115.505,-40.540,178.887,5.723,149.346
C06293=1176.099,-115.755,-40.532,178.885,5.722,149.347
C06294=1176.105,-116.004,-40.522,178.883,5.722,149.347
C06295=1176.110,-116.254,-40.513,178.881,5.721,149.348
C06296=1176.115,-116.504,-40.504,178.879,5.722,149.349
C06297=1176.120,-116.753,-40.495,178.877,5.721,149.349
C06298=1176.125,-117.003,-40.486,178.875,5.722,149.350
C06299=1176.131,-117.253,-40.477,178.872,5.721,149.350
C06300=1176.137,-117.503,-40.468,178.871,5.721,149.351
C06301=1176.142,-117.753,-40.459,178.868,5.720,149.352
C06302=1176.147,-118.003,-40.450,178.866,5.720,149.352
C06303=1176.152,-118.253,-40.441,178.864,5.720,149.353
C06304=1176.158,-118.502,-40.433,178.862,5.720,149.353
C06305=1176.163,-118.752,-40.424,178.859,5.720,149.354
C06306=1176.169,-119.002,-40.414,178.858,5.720,149.354
C06307=1176.174,-119.252,-40.405,178.856,5.719,149.355
C06308=1176.179,-119.502,-40.396,178.854,5.719,149.356
C06309=1176.184,-119.751,-40.387,178.851,5.719,149.356
C06310=1176.189,-120.001,-40.378,178.850,5.719,149.357
C06311=1176.195,-120.250,-40.369,178.847,5.718,149.357
C06312=1176.200,-120.500,-40.360,178.846,5.718,149.358
C06313=1176.205,-120.750,-40.352,178.843,5.718,149.359
C06314=1176.211,-121.000,-40.342,178.841,5.718,149.359
C06315=1176.216,-121.250,-40.333,178.839,5.717,149.359
C06316=1176.222,-121.500,-40.325,178.837,5.718,149.360
C06317=1176.227,-121.750,-40.316,178.835,5.717,149.361
C06318=1176.233,-121.999,-40.308,178.833,5.717,149.361
C06319=1176.238,-122.249,-40.299,178.831,5.716,149.362
C06320=1176.243,-122.499,-40.290,178.829,5.717,149.362
C06321=1176.248,-122.749,-40.281,178.826,5.716,149.363
C06322=1176.253,-122.999,-40.272,178.825,5.716,149.364
C06323=1176.259,-123.248,-40.263,178.822,5.716,149.364
C06324=1176.264,-123.498,-40.254,178.820,5.716,149.365
C06325=1176.270,-123.747,-40.246,178.818,5.715,149.365
C06326=1176.275,-123.997,-40.237,178.816,5.715,149.366
C06327=1176.281,-124.247,-40.227,178.814,5.715,149.366
C06328=1176.286,-124.497,-40.218,178.812,5.715,149.367
C06329=1176.292,-124.746,-40.210,178.810,5.714,149.368
C06330=1176.297,-124.997,-40.202,178.808,5.714,149.368
C06331=1176.302,-125.247,-40.193,178.806,5.715,149.369
C06332=1176.307,-125.497,-40.184,178.804,5.714,149.369
C06333=1176.313,-125.746,-40.175,178.802,5.714,149.370
C06334=1176.318,-125.996,-40.166,178.799,5.714,149.371
C06335=1176.323,-126.245,-40.157,178.798,5.714,149.371
C06336=1176.329,-126.495,-40.149,178.796,5.713,149.372
C06337=1176.334,-126.745,-40.140,178.794,5.713,149.372
C06338=1176.340,-126.995,-40.132,178.791,5.713,149.373
C06339=1176.345,-127.245,-40.123,178.790,5.713,149.373
C06340=1176.350,-127.495,-40.114,178.787,5.712,149.374
C06341=1175.929,-127.505,-40.154,178.783,5.716,149.376
C06342=1175.923,-127.256,-40.163,178.786,5.716,149.375
C06343=1175.918,-127.006,-40.172,178.787,5.716,149.375
C06344=1175.913,-126.756,-40.181,178.790,5.717,149.374
C06345=1175.908,-126.507,-40.190,178.792,5.716,149.373
C06346=1175.902,-126.256,-40.198,178.794,5.717,149.373
C06347=1175.897,-126.007,-40.206,178.796,5.717,149.372
C06348=1175.891,-125.757,-40.215,178.798,5.717,149.372
C06349=1175.886,-125.507,-40.224,178.800,5.717,149.371
C06350=1175.881,-125.257,-40.233,178.802,5.718,149.371
C06351=1175.875,-125.008,-40.242,178.804,5.718,149.370
C06352=1175.870,-124.758,-40.251,178.806,5.718,149.370
C06353=1175.865,-124.508,-40.259,178.808,5.718,149.369
C06354=1175.860,-124.258,-40.268,178.811,5.719,149.368
C06355=1175.854,-124.008,-40.277,178.812,5.719,149.368
C06356=1175.848,-123.759,-40.286,178.815,5.719,149.367
C06357=1175.843,-123.509,-40.295,178.816,5.719,149.367
C06358=1175.837,-123.259,-40.303,178.819,5.720,149.366
C06359=1175.832,-123.009,-40.312,178.821,5.719,149.365
C06360=1175.827,-122.759,-40.321,178.823,5.720,149.365
C06361=1175.822,-122.509,-40.330,178.825,5.720,149.364
C06362=1175.816,-122.260,-40.339,178.827,5.721,149.364
C06363=1175.811,-122.010,-40.348,178.829,5.720,149.363
C06364=1175.806,-121.761,-40.356,178.832,5.721,149.363
C06365=1175.801,-121.511,-40.365,178.833,5.721,149.362
C06366=1175.796,-121.261,-40.374,178.835,5.722,149.362
C06367=1175.790,-121.011,-40.383,178.837,5.721,149.361
C06368=1175.785,-120.762,-40.392,178.840,5.722,149.360
C06369=1175.779,-120.512,-40.401,178.842,5.722,149.360
C06370=1175.774,-120.262,-40.410,178.844,5.722,149.359
C06371=1175.768,-120.012,-40.419,178.845,5.722,149.359
C06372=1175.763,-119.762,-40.428,178.848,5.723,149.358
C06373=1175.758,-119.512,-40.437,178.850,5.723,149.357
C06374=1175.753,-119.262,-40.446,178.852,5.723,149.357
C06375=1175.747,-119.013,-40.454,178.854,5.723,149.356
C06376=1175.742,-118.763,-40.463,178.856,5.724,149.356
C06377=1175.736,-118.513,-40.473,178.858,5.723,149.355
C06378=1175.731,-118.263,-40.482,178.860,5.724,149.355
C06379=1175.726,-118.014,-40.490,178.863,5.724,149.354
C06380=1175.721,-117.764,-40.499,178.865,5.724,149.353
C06381=1175.715,-117.514,-40.508,178.866,5.724,149.353
C06382=1175.710,-117.264,-40.517,178.869,5.725,149.352
C06383=1175.704,-117.015,-40.526,178.871,5.725,149.352
C06384=1175.699,-116.765,-40.535,178.873,5.725,149.351
C06385=1175.693,-116.515,-40.544,178.875,5.725,149.350
C06386=1175.688,-116.265,-40.553,178.877,5.726,149.350
C06387=1175.683,-116.016,-40.563,178.879,5.725,149.349
C06388=1175.678,-115.766,-40.571,178.881,5.726,149.349
C06389=1175.672,-115.516,-40.581,178.883,5.726,149.348
C06390=1175.667,-115.266,-40.590,178.886,5.727,149.348
C06391=1175.662,-115.016,-40.599,178.887,5.727,149.347
C06392=1175.657,-114.766,-40.608,178.890,5.727,149.346
C06393=1175.651,-114.516,-40.617,178.892,5.727,149.346
C06394=1175.645,-114.267,-40.626,178.894,5.727,149.345
C06395=1175.640,-114.018,-40.635,178.896,5.727,149.345
C06396=1175.635,-113.768,-40.644,178.898,5.728,149.344
C06397=1175.630,-113.518,-40.653,178.900,5.728,149.344
C06398=1175.624,-113.268,-40.663,178.902,5.728,149.343
C06399=1175.619,-113.018,-40.671,178.904,5.728,149.342
C06400=1175.614,-112.768,-40.680,178.907,5.729,149.342
C06401=1175.609,-112.519,-40.690,178.909,5.728,149.341
C06402=1175.603,-112.269,-40.699,178.911,5.729,149.341
C06403=1175.598,-112.019,-40.708,178.914,5.730,149.340
C06404=1175.593,-111.769,-40.717,178.915,5.729,149.339
C06405=1175.587,-111.519,-40.727,178.917,5.730,149.339
C06406=1175.582,-111.270,-40.736,178.919,5.730,149.338
C06407=1175.577,-111.020,-40.745,178.922,5.731,149.338
C06408=1175.571,-110.770,-40.754,178.924,5.730,149.337
C06409=1175.566,-110.520,-40.764,178.926,5.731,149.337
C06410=1175.561,-110.271,-40.773,178.928,5.731,149.336
C06411=1175.556,-110.021,-40.782,178.930,5.731,149.335
C06412=1175.550,-109.771,-40.792,178.932,5.731,149.335
C06413=1175.544,-109.521,-40.801,178.934,5.732,149.334
C06414=1175.540,-109.271,-40.810,178.936,5.732,149.334
C06415=1175.534,-109.021,-40.820,178.939,5.732,149.333
C06416=1175.529,-108.771,-40.829,178.940,5.732,149.332
C06417=1175.524,-108.522,-40.838,178.943,5.732,149.332
C06418=1175.518,-108.272,-40.848,178.945,5.733,149.331
C06419=1175.513,-108.022,-40.857,178.947,5.733,149.331
C06420=1175.508,-107.773,-40.866,178.949,5.734,149.330
C06421=1175.502,-107.523,-40.876,178.951,5.734,149.330
C06422=1175.497,-107.273,-40.885,178.954,5.734,149.329
C06423=1175.492,-107.024,-40.894,178.955,5.734,149.328
C06424=1175.486,-106.774,-40.904,178.958,5.734,149.328
C06425=1175.481,-106.524,-40.913,178.960,5.734,149.327
C06426=1175.476,-106.274,-40.922,178.962,5.735,149.326
C06427=1175.470,-106.024,-40.932,178.964,5.735,149.326
C06428=1175.465,-105.774,-40.941,178.967,5.735,149.325
C06429=1175.459,-105.525,-40.951,178.969,5.736,149.325
C06430=1175.454,-105.275,-40.960,178.971,5.735,149.324
C06431=1175.449,-105.026,-40.969,178.973,5.736,149.324
C06432=1175.443,-104.776,-40.979,178.975,5.736,149.323
C06433=1175.438,-104.526,-40.988,178.977,5.737,149.322
C06434=1175.433,-104.276,-40.998,178.979,5.737,149.322
C06435=1175.427,-104.026,-41.007,178.982,5.737,149.321
C06436=1175.423,-103.777,-41.016,178.983,5.737,149.321
C06437=1175.417,-103.527,-41.026,178.986,5.737,149.320
C06438=1175.411,-103.277,-41.035,178.988,5.738,149.319
C06439=1175.406,-103.028,-41.045,178.990,5.738,149.319
C06440=1175.401,-102.777,-41.054,178.992,5.738,149.318
C06441=1175.396,-102.528,-41.064,178.994,5.738,149.318
C06442=1175.390,-102.256,-41.074,178.997,5.739,149.317
C06443=1175.384,-101.984,-41.085,178.999,5.739,149.316
C06444=1175.379,-101.712,-41.095,179.001,5.739,149.316
C06445=1175.372,-101.440,-41.106,179.003,5.740,149.315
C06446=1175.368,-101.191,-41.115,179.006,5.740,149.314
C06447=1175.362,-100.941,-41.124,179.008,5.740,149.314
C06448=1175.357,-100.692,-41.134,179.010,5.740,149.313
C06449=1175.352,-100.442,-41.143,179.012,5.740,149.313
C06450=1175.346,-100.192,-41.153,179.015,5.741,149.312
C06451=1175.341,-99.942,-41.162,179.016,5.741,149.312
C06452=1175.336,-99.692,-41.173,179.019,5.741,149.311
C06453=1175.331,-99.442,-41.182,179.021,5.742,149.310
C06454=1175.325,-99.193,-41.192,179.023,5.741,149.310
C06455=1175.320,-98.943,-41.202,179.025,5.742,149.309
C06456=1175.314,-98.693,-41.211,179.028,5.742,149.308
C06457=1175.309,-98.444,-41.221,179.030,5.743,149.308
C06458=1175.304,-98.194,-41.230,179.032,5.742,149.307
C06459=1175.298,-97.944,-41.240,179.034,5.743,149.307
C06460=1175.293,-97.694,-41.250,179.037,5.743,149.306
C06461=1175.288,-97.444,-41.260,179.038,5.743,149.306
C06462=1175.283,-97.195,-41.270,179.041,5.744,149.305
C06463=1175.277,-96.945,-41.279,179.043,5.744,149.304
C06464=1175.272,-96.696,-41.289,179.045,5.744,149.304
C06465=1175.266,-96.445,-41.298,179.047,5.744,149.303
C06466=1175.261,-96.196,-41.308,179.049,5.744,149.302
C06467=1175.256,-95.946,-41.318,179.052,5.745,149.302
C06468=1175.250,-95.696,-41.328,179.054,5.745,149.301
C06469=1175.246,-95.447,-41.337,179.056,5.746,149.301
C06470=1175.240,-95.197,-41.348,179.058,5.745,149.300
C06471=1175.235,-94.947,-41.357,179.060,5.746,149.300
C06472=1175.229,-94.698,-41.367,179.063,5.746,149.299
C06473=1175.224,-94.447,-41.377,179.064,5.746,149.298
C06474=1175.219,-94.198,-41.386,179.067,5.747,149.298
C06475=1175.213,-93.948,-41.396,179.069,5.747,149.297
C06476=1175.209,-93.699,-41.406,179.071,5.747,149.297
C06477=1175.203,-93.449,-41.416,179.073,5.747,149.296
C06478=1175.198,-93.198,-41.426,179.076,5.747,149.295
C06479=1175.193,-92.949,-41.436,179.078,5.748,149.295
C06480=1175.187,-92.700,-41.446,179.080,5.748,149.294
C06481=1175.181,-92.449,-41.455,179.082,5.749,149.294
C06482=1175.177,-92.200,-41.465,179.084,5.748,149.293
C06483=1175.172,-91.950,-41.476,179.086,5.749,149.292
C06484=1175.166,-91.700,-41.485,179.089,5.749,149.292
C06485=1175.161,-91.451,-41.495,179.091,5.749,149.291
C06486=1175.155,-91.201,-41.505,179.093,5.750,149.291
C06487=1175.150,-90.951,-41.515,179.095,5.750,149.290
C06488=1175.145,-90.702,-41.525,179.098,5.750,149.289
C06489=1175.139,-90.451,-41.535,179.100,5.751,149.289
C06490=1175.134,-90.202,-41.545,179.102,5.751,149.288
C06491=1175.129,-89.953,-41.554,179.104,5.751,149.288
C06492=1175.124,-89.702,-41.565,179.106,5.751,149.287
C06493=1175.118,-89.453,-41.575,179.108,5.752,149.286
C06494=1175.113,-89.203,-41.584,179.111,5.752,149.286
C06495=1175.108,-88.953,-41.595,179.113,5.752,149.285
C06496=1175.103,-88.703,-41.605,179.115,5.753,149.285
C06497=1175.097,-88.454,-41.615,179.118,5.753,149.284
C06498=1175.092,-88.204,-41.625,179.120,5.753,149.283
C06499=1175.087,-87.954,-41.635,179.122,5.754,149.283
C06500=1175.081,-87.704,-41.645,179.124,5.753,149.282
C06501=1175.076,-87.455,-41.654,179.127,5.754,149.281
C06502=1175.071,-87.205,-41.665,179.129,5.754,149.281
C06503=1175.066,-86.955,-41.675,179.131,5.754,149.280
C06504=1175.060,-86.705,-41.685,179.133,5.755,149.280
C06505=1175.055,-86.456,-41.695,179.135,5.754,149.279
C06506=1175.050,-86.206,-41.706,179.137,5.755,149.279
C06507=1175.045,-85.956,-41.716,179.140,5.756,149.278
C06508=1175.039,-85.706,-41.725,179.142,5.756,149.277
C06509=1175.034,-85.456,-41.736,179.144,5.756,149.277
C06510=1175.029,-85.207,-41.745,179.146,5.757,149.276
C06511=1175.023,-84.957,-41.756,179.148,5.756,149.276
C06512=1175.018,-84.708,-41.766,179.151,5.757,149.275
C06513=1175.013,-84.457,-41.776,179.153,5.757,149.274
C06514=1175.008,-84.208,-41.786,179.155,5.758,149.274
C06515=1175.002,-83.959,-41.796,179.158,5.758,149.273
C06516=1174.997,-83.708,-41.807,179.160,5.758,149.272
C06517=1174.992,-83.459,-41.817,179.162,5.758,149.272
C06518=1174.986,-83.209,-41.827,179.165,5.759,149.271
C06519=1174.981,-82.959,-41.838,179.166,5.759,149.271
C06520=1174.976,-82.710,-41.847,179.169,5.759,149.270
C06521=1174.971,-82.460,-41.858,179.170,5.759,149.270
C06522=1174.966,-82.210,-41.868,179.173,5.760,149.269
C06523=1174.960,-81.961,-41.878,179.175,5.760,149.268
C06524=1174.955,-81.710,-41.889,179.177,5.760,149.268
C06525=1174.949,-81.461,-41.899,179.180,5.761,149.267
C06526=1174.944,-81.211,-41.909,179.182,5.761,149.266
C06527=1174.940,-80.961,-41.919,179.184,5.761,149.266
C06528=1174.934,-80.712,-41.930,179.186,5.762,149.265
C06529=1174.928,-80.462,-41.940,179.189,5.762,149.265
C06530=1174.923,-80.212,-41.950,179.191,5.762,149.264
C06531=1174.918,-79.962,-41.961,179.193,5.762,149.263
C06532=1174.912,-79.713,-41.971,179.195,5.762,149.263
C06533=1174.907,-79.463,-41.982,179.198,5.763,149.262
C06534=1174.902,-79.214,-41.992,179.200,5.764,149.262
C06535=1174.897,-78.963,-42.003,179.202,5.763,149.261
C06536=1174.892,-78.714,-42.013,179.204,5.764,149.261
C06537=1174.886,-78.465,-42.023,179.207,5.764,149.260
C06538=1174.881,-78.214,-42.033,179.209,5.764,149.259
C06539=1174.876,-77.965,-42.043,179.211,5.765,149.259
C06540=1174.871,-77.715,-42.054,179.214,5.765,149.258
C06541=1174.865,-77.465,-42.064,179.215,5.765,149.257
C06542=1174.860,-77.216,-42.075,179.218,5.765,149.257
C06543=1174.855,-76.966,-42.086,179.220,5.766,149.256
C06544=1174.849,-76.716,-42.096,179.222,5.766,149.256
C06545=1174.844,-76.466,-42.107,179.225,5.766,149.255
C06546=1174.838,-76.195,-42.118,179.227,5.767,149.254
C06547=1174.833,-75.925,-42.129,179.230,5.767,149.254
C06548=1174.827,-75.653,-42.141,179.232,5.767,149.253
C06549=1174.821,-75.382,-42.151,179.235,5.767,149.252
C06550=1174.817,-75.133,-42.163,179.237,5.768,149.252
C06551=1174.811,-74.883,-42.173,179.239,5.769,149.251
C06552=1174.806,-74.633,-42.184,179.241,5.769,149.251
C06553=1174.800,-74.383,-42.194,179.244,5.769,149.250
C06554=1174.795,-74.133,-42.204,179.245,5.769,149.249
C06555=1174.790,-73.884,-42.215,179.248,5.769,149.249
C06556=1174.784,-73.635,-42.225,179.251,5.770,149.248
C06557=1174.779,-73.384,-42.236,179.253,5.771,149.247
C06558=1174.774,-73.135,-42.246,179.255,5.770,149.247
C06559=1174.768,-72.885,-42.258,179.257,5.771,149.246
C06560=1174.763,-72.635,-42.268,179.260,5.771,149.246
C06561=1174.758,-72.385,-42.279,179.261,5.771,149.245
C06562=1174.752,-72.136,-42.289,179.264,5.772,149.244
C06563=1174.748,-71.886,-42.300,179.267,5.772,149.244
C06564=1174.742,-71.636,-42.311,179.268,5.772,149.243
C06565=1174.737,-71.386,-42.321,179.271,5.773,149.242
C06566=1174.732,-71.137,-42.332,179.273,5.774,149.242
C06567=1174.727,-70.887,-42.343,179.275,5.773,149.241
C06568=1174.721,-70.638,-42.353,179.278,5.774,149.241
C06569=1174.716,-70.388,-42.364,179.280,5.774,149.240
C06570=1174.711,-70.138,-42.374,179.282,5.774,149.239
C06571=1174.706,-69.888,-42.385,179.284,5.775,149.239
C06572=1174.700,-69.639,-42.397,179.287,5.775,149.238
C06573=1174.695,-69.389,-42.407,179.289,5.775,149.238
C06574=1174.689,-69.140,-42.418,179.291,5.776,149.237
C06575=1174.684,-68.889,-42.429,179.294,5.776,149.236
C06576=1174.679,-68.640,-42.439,179.296,5.776,149.236
C06577=1174.674,-68.390,-42.450,179.298,5.776,149.235
C06578=1174.669,-68.141,-42.460,179.300,5.777,149.235
C06579=1174.664,-67.891,-42.472,179.303,5.778,149.234
C06580=1174.658,-67.641,-42.483,179.305,5.778,149.233
C06581=1174.653,-67.391,-42.493,179.307,5.778,149.233
C06582=1174.648,-67.141,-42.504,179.310,5.778,149.232
C06583=1174.642,-66.892,-42.514,179.312,5.778,149.232
C06584=1174.638,-66.642,-42.526,179.314,5.779,149.231
C06585=1174.632,-66.393,-42.536,179.316,5.780,149.230
C06586=1174.627,-66.143,-42.547,179.319,5.779,149.230
C06587=1174.621,-65.893,-42.558,179.321,5.780,149.229
C06588=1174.616,-65.644,-42.569,179.323,5.780,149.228
C06589=1174.611,-65.393,-42.580,179.325,5.780,149.228
C06590=1174.606,-65.144,-42.591,179.328,5.781,149.227
C06591=1174.601,-64.894,-42.601,179.330,5.781,149.227
C06592=1174.595,-64.645,-42.613,179.333,5.782,149.226
C06593=1174.590,-64.395,-42.624,179.335,5.782,149.225
C06594=1174.585,-64.145,-42.635,179.337,5.782,149.225
C06595=1174.580,-63.896,-42.645,179.339,5.783,149.224
C06596=1174.575,-63.646,-42.656,179.342,5.782,149.224
C06597=1174.569,-63.396,-42.667,179.344,5.783,149.223
C06598=1174.564,-63.146,-42.678,179.346,5.784,149.222
C06599=1174.559,-62.896,-42.689,179.349,5.784,149.222
C06600=1174.554,-62.647,-42.700,179.351,5.784,149.221
C06601=1174.548,-62.397,-42.711,179.353,5.785,149.220
C06602=1174.543,-62.148,-42.722,179.356,5.785,149.220
C06603=1174.538,-61.898,-42.733,179.358,5.785,149.219
C06604=1174.533,-61.648,-42.744,179.360,5.785,149.219
C06605=1174.527,-61.399,-42.755,179.362,5.786,149.218
C06606=1174.522,-61.148,-42.766,179.365,5.787,149.217
C06607=1174.517,-60.899,-42.777,179.367,5.787,149.217
C06608=1174.511,-60.650,-42.789,179.369,5.787,149.216
C06609=1174.506,-60.399,-42.799,179.372,5.787,149.215
C06610=1174.501,-60.150,-42.811,179.374,5.788,149.215
C06611=1174.496,-59.901,-42.822,179.376,5.788,149.214
C06612=1174.490,-59.650,-42.833,179.379,5.788,149.214
C06613=1174.486,-59.401,-42.844,179.381,5.789,149.213
C06614=1174.480,-59.151,-42.854,179.383,5.789,149.212
C06615=1174.475,-58.901,-42.866,179.385,5.789,149.212
C06616=1174.470,-58.651,-42.877,179.388,5.790,149.211
C06617=1174.465,-58.403,-42.888,179.391,5.790,149.211
C06618=1174.459,-58.152,-42.899,179.392,5.790,149.210
C06619=1174.454,-57.902,-42.911,179.395,5.791,149.209
C06620=1174.449,-57.653,-42.922,179.397,5.791,149.209
C06621=1174.443,-57.403,-42.933,179.400,5.792,149.208
C06622=1174.439,-57.153,-42.944,179.402,5.792,149.207
C06623=1174.433,-56.904,-42.955,179.404,5.792,149.207
C06624=1174.428,-56.654,-42.967,179.407,5.793,149.206
C06625=1174.423,-56.404,-42.978,179.409,5.794,149.206
C06626=1174.418,-56.155,-42.989,179.411,5.793,149.205
C06627=1174.412,-55.905,-43.000,179.414,5.794,149.204
C06628=1174.407,-55.656,-43.012,179.416,5.794,149.204
C06629=1174.402,-55.405,-43.023,179.419,5.795,149.203
C06630=1174.397,-55.155,-43.034,179.420,5.795,149.203
C06631=1174.392,-54.907,-43.045,179.423,5.795,149.202
C06632=1174.386,-54.657,-43.057,179.426,5.796,149.201
C06633=1174.382,-54.407,-43.068,179.428,5.796,149.201
C06634=1174.375,-54.157,-43.079,179.430,5.796,149.200
C06635=1174.371,-53.908,-43.090,179.432,5.796,149.199
C06636=1174.366,-53.658,-43.102,179.435,5.797,149.199
C06637=1174.360,-53.408,-43.113,179.437,5.798,149.198
C06638=1174.356,-53.158,-43.125,179.439,5.798,149.198
C06639=1174.350,-52.909,-43.136,179.442,5.798,149.197
C06640=1174.345,-52.659,-43.147,179.444,5.799,149.196
C06641=1174.339,-52.409,-43.159,179.446,5.799,149.196
C06642=1174.335,-52.159,-43.170,179.448,5.799,149.195
C06643=1174.329,-51.910,-43.182,179.451,5.800,149.195
C06644=1174.324,-51.660,-43.193,179.453,5.800,149.194
C06645=1174.319,-51.411,-43.204,179.456,5.801,149.193
C06646=1174.314,-51.161,-43.216,179.458,5.801,149.193
C06647=1174.309,-50.912,-43.227,179.460,5.801,149.192
C06648=1174.303,-50.662,-43.239,179.463,5.801,149.191
C06649=1174.298,-50.412,-43.249,179.465,5.802,149.191
C06650=1174.293,-50.141,-43.262,179.468,5.803,149.190
C06651=1174.287,-49.871,-43.274,179.470,5.803,149.190
C06652=1174.281,-49.601,-43.287,179.472,5.803,149.189
C06653=1174.276,-49.330,-43.299,179.475,5.803,149.188
C06654=1174.270,-49.081,-43.311,179.477,5.804,149.188
C06655=1174.265,-48.831,-43.322,179.480,5.804,149.187
C06656=1174.259,-48.581,-43.334,179.482,5.805,149.186
C06657=1174.255,-48.331,-43.345,179.484,5.805,149.186
C06658=1174.249,-48.081,-43.357,179.487,5.805,149.185
C06659=1174.243,-47.832,-43.369,179.489,5.806,149.185
C06660=1174.239,-47.583,-43.380,179.492,5.807,149.184
C06661=1174.233,-47.333,-43.392,179.494,5.807,149.183
C06662=1174.229,-47.083,-43.403,179.496,5.807,149.183
C06663=1174.223,-46.833,-43.415,179.499,5.807,149.182
C06664=1174.218,-46.583,-43.426,179.501,5.808,149.182
C06665=1174.212,-46.334,-43.438,179.504,5.809,149.181
C06666=1174.207,-46.085,-43.451,179.506,5.809,149.180
C06667=1174.203,-45.835,-43.462,179.508,5.809,149.180
C06668=1174.197,-45.585,-43.474,179.510,5.809,149.179
C06669=1174.192,-45.336,-43.485,179.513,5.810,149.179
C06670=1174.187,-45.086,-43.497,179.515,5.811,149.178
C06671=1174.182,-44.836,-43.509,179.518,5.811,149.177
C06672=1174.176,-44.587,-43.520,179.520,5.811,149.177
C06673=1174.171,-44.337,-43.532,179.522,5.812,149.176
C06674=1174.165,-44.087,-43.544,179.525,5.812,149.175
C06675=1174.161,-43.837,-43.555,179.527,5.813,149.175
C06676=1174.155,-43.587,-43.567,179.530,5.813,149.174
C06677=1174.151,-43.338,-43.579,179.532,5.813,149.173
C06678=1174.145,-43.089,-43.591,179.534,5.814,149.173
C06679=1174.140,-42.839,-43.602,179.537,5.814,149.172
C06680=1174.135,-42.589,-43.614,179.539,5.815,149.172
C06681=1174.130,-42.339,-43.626,179.542,5.815,149.171
C06682=1174.124,-42.090,-43.637,179.544,5.815,149.170
C06683=1174.119,-41.841,-43.650,179.546,5.816,149.170
C06684=1174.114,-41.591,-43.661,179.548,5.816,149.169
C06685=1174.109,-41.341,-43.673,179.551,5.817,149.168
C06686=1174.103,-41.091,-43.685,179.553,5.817,149.168
C06687=1174.099,-40.841,-43.696,179.555,5.817,149.167
C06688=1174.093,-40.592,-43.709,179.558,5.818,149.167
C06689=1174.088,-40.342,-43.721,179.560,5.818,149.166
C06690=1174.083,-40.092,-43.732,179.563,5.819,149.165
C06691=1174.078,-39.843,-43.744,179.565,5.820,149.165
C06692=1174.073,-39.593,-43.756,179.567,5.819,149.164
C06693=1174.067,-39.343,-43.768,179.570,5.820,149.163
C06694=1174.063,-39.094,-43.780,179.572,5.820,149.163
C06695=1174.057,-38.844,-43.791,179.575,5.821,149.162
C06696=1174.052,-38.594,-43.804,179.577,5.821,149.162
C06697=1174.046,-38.345,-43.816,179.580,5.822,149.161
C06698=1174.041,-38.096,-43.827,179.582,5.822,149.160
C06699=1174.036,-37.846,-43.839,179.584,5.823,149.160
C06700=1174.031,-37.596,-43.851,179.586,5.823,149.159
C06701=1174.025,-37.346,-43.863,179.589,5.823,149.159
C06702=1174.020,-37.096,-43.875,179.591,5.824,149.158
C06703=1174.016,-36.847,-43.887,179.594,5.825,149.157
C06704=1174.010,-36.598,-43.899,179.596,5.824,149.157
C06705=1174.005,-36.348,-43.911,179.598,5.825,149.156
C06706=1174.000,-36.098,-43.924,179.601,5.826,149.156
C06707=1173.994,-35.848,-43.935,179.604,5.826,149.155
C06708=1173.989,-35.598,-43.947,179.606,5.827,149.154
C06709=1173.984,-35.349,-43.959,179.608,5.827,149.154
C06710=1173.979,-35.099,-43.971,179.610,5.827,149.153
C06711=1173.974,-34.850,-43.984,179.613,5.828,149.152
C06712=1173.968,-34.600,-43.996,179.615,5.828,149.152
C06713=1173.963,-34.350,-44.008,179.617,5.829,149.151
C06714=1173.958,-34.101,-44.020,179.620,5.829,149.151
C06715=1173.953,-33.851,-44.031,179.623,5.830,149.150
C06716=1173.948,-33.602,-44.044,179.625,5.831,149.149
C06717=1173.943,-33.352,-44.056,179.627,5.830,149.149
C06718=1173.938,-33.102,-44.069,179.630,5.831,149.148
C06719=1173.933,-32.852,-44.081,179.632,5.831,149.148
C06720=1173.927,-32.603,-44.093,179.635,5.832,149.147
C06721=1173.922,-32.353,-44.105,179.637,5.833,149.146
C06722=1173.917,-32.103,-44.117,179.639,5.833,149.146
C06723=1173.911,-31.854,-44.130,179.641,5.833,149.145
C06724=1173.907,-31.604,-44.141,179.644,5.834,149.145
C06725=1173.902,-31.355,-44.154,179.646,5.834,149.144
C06726=1173.896,-31.105,-44.166,179.649,5.835,149.143
C06727=1173.891,-30.855,-44.178,179.651,5.835,149.143
C06728=1173.886,-30.606,-44.191,179.654,5.836,149.142
C06729=1173.881,-30.356,-44.203,179.656,5.836,149.141
C06730=1173.875,-30.107,-44.215,179.659,5.837,149.141
C06731=1173.870,-29.857,-44.227,179.661,5.837,149.140
C06732=1173.865,-29.607,-44.240,179.663,5.837,149.139
C06733=1173.860,-29.357,-44.252,179.666,5.838,149.139
C06734=1173.855,-29.108,-44.265,179.668,5.838,149.138
C06735=1173.849,-28.858,-44.276,179.670,5.839,149.138
C06736=1173.844,-28.608,-44.289,179.673,5.840,149.137
C06737=1173.839,-28.359,-44.302,179.676,5.840,149.136
C06738=1173.834,-28.109,-44.314,179.677,5.840,149.136
C06739=1173.829,-27.860,-44.326,179.680,5.841,149.135
C06740=1173.823,-27.610,-44.338,179.683,5.841,149.135
C06741=1173.819,-27.360,-44.351,179.685,5.842,149.134
C06742=1173.814,-27.110,-44.364,179.687,5.842,149.133
C06743=1173.808,-26.861,-44.375,179.690,5.843,149.133
C06744=1173.803,-26.611,-44.388,179.692,5.843,149.132
C06745=1173.798,-26.362,-44.401,179.695,5.844,149.131
C06746=1173.792,-26.112,-44.413,179.698,5.844,149.131
C06747=1173.787,-25.863,-44.425,179.699,5.844,149.130
C06748=1173.783,-25.613,-44.438,179.702,5.845,149.130
C06749=1173.777,-25.363,-44.450,179.704,5.846,149.129
C06750=1173.772,-25.113,-44.463,179.707,5.846,149.128
C06751=1173.767,-24.864,-44.475,179.709,5.847,149.128
C06752=1173.762,-24.614,-44.487,179.712,5.847,149.127
C06753=1173.757,-24.365,-44.500,179.714,5.848,149.127
C06754=1173.752,-24.095,-44.513,179.717,5.848,149.126
C06755=1173.746,-23.825,-44.528,179.720,5.849,149.125
C06756=1173.740,-23.555,-44.540,179.722,5.849,149.124
C06757=1173.734,-23.285,-44.555,179.725,5.850,149.124
C06758=1173.729,-23.036,-44.567,179.727,5.850,149.123
C06759=1173.724,-22.787,-44.580,179.730,5.851,149.123
C06760=1173.719,-22.536,-44.592,179.732,5.852,149.122
C06761=1173.714,-22.287,-44.605,179.735,5.852,149.121
C06762=1173.709,-22.037,-44.617,179.737,5.852,149.121
C06763=1173.704,-21.788,-44.630,179.739,5.853,149.120
C06764=1173.698,-21.538,-44.642,179.741,5.853,149.120
C06765=1173.693,-21.288,-44.655,179.744,5.853,149.119
C06766=1173.688,-21.039,-44.668,179.746,5.854,149.118
C06767=1173.683,-20.789,-44.680,179.749,5.855,149.118
C06768=1173.678,-20.540,-44.693,179.752,5.855,149.117
C06769=1173.673,-20.290,-44.706,179.754,5.856,149.117
C06770=1173.668,-20.040,-44.718,179.756,5.856,149.116
C06771=1173.662,-19.790,-44.731,179.759,5.857,149.115
C06772=1173.657,-19.541,-44.744,179.761,5.858,149.115
C06773=1173.652,-19.292,-44.756,179.764,5.858,149.114
C06774=1173.647,-19.042,-44.769,179.766,5.858,149.114
C06775=1173.642,-18.792,-44.782,179.768,5.859,149.113
C06776=1173.636,-18.543,-44.795,179.771,5.859,149.112
C06777=1173.631,-18.293,-44.808,179.773,5.860,149.112
C06778=1173.627,-18.043,-44.821,179.776,5.860,149.111
C06779=1173.621,-17.794,-44.833,179.778,5.861,149.110
C06780=1173.616,-17.544,-44.845,179.780,5.862,149.110
C06781=1173.611,-17.294,-44.859,179.783,5.862,149.109
C06782=1173.606,-17.044,-44.871,179.786,5.862,149.108
C06783=1173.600,-16.795,-44.884,179.788,5.863,149.108
C06784=1173.595,-16.546,-44.896,179.791,5.864,149.107
C06785=1173.590,-16.296,-44.910,179.793,5.864,149.107
C06786=1173.585,-16.046,-44.923,179.795,5.865,149.106
C06787=1173.580,-15.797,-44.935,179.798,5.865,149.105
C06788=1173.575,-15.547,-44.948,179.800,5.865,149.105
C06789=1173.569,-15.297,-44.961,179.802,5.866,149.104
C06790=1173.564,-15.048,-44.974,179.805,5.866,149.104
C06791=1173.560,-14.798,-44.987,179.807,5.867,149.103
C06792=1173.554,-14.548,-45.000,179.810,5.868,149.102
C06793=1173.549,-14.299,-45.013,179.813,5.868,149.102
C06794=1173.544,-14.049,-45.026,179.815,5.869,149.101
C06795=1173.538,-13.799,-45.039,179.817,5.869,149.101
C06796=1173.534,-13.551,-45.052,179.820,5.870,149.100
C06797=1173.529,-13.301,-45.065,179.822,5.871,149.099
C06798=1173.524,-13.051,-45.078,179.825,5.871,149.099
C06799=1173.518,-12.802,-45.091,179.828,5.872,149.098
C06800=1173.514,-12.552,-45.104,179.830,5.872,149.098
C06801=1173.508,-12.302,-45.117,179.832,5.873,149.097
C06802=1173.503,-12.053,-45.130,179.835,5.873,149.096
C06803=1173.498,-11.803,-45.143,179.837,5.874,149.096
C06804=1173.492,-11.553,-45.156,179.840,5.875,149.095
C06805=1173.487,-11.304,-45.169,179.843,5.875,149.094
C06806=1173.483,-11.054,-45.182,179.845,5.876,149.094
C06807=1173.477,-10.805,-45.195,179.847,5.876,149.093
C06808=1173.472,-10.555,-45.208,179.850,5.877,149.093
C06809=1173.467,-10.305,-45.221,179.852,5.877,149.092
C06810=1173.461,-10.056,-45.234,179.854,5.877,149.091
C06811=1173.457,-9.806,-45.248,179.856,5.878,149.091
C06812=1173.451,-9.557,-45.261,179.859,5.879,149.090
C06813=1173.447,-9.307,-45.274,179.862,5.879,149.089
C06814=1173.442,-9.057,-45.287,179.864,5.880,149.089
C06815=1173.436,-8.808,-45.300,179.867,5.880,149.088
C06816=1173.432,-8.558,-45.313,179.869,5.881,149.088
C06817=1173.426,-8.309,-45.327,179.871,5.882,149.087
C06818=1173.421,-8.059,-45.340,179.874,5.882,149.086
C06819=1173.415,-7.809,-45.353,179.877,5.883,149.086
C06820=1173.411,-7.560,-45.367,179.879,5.883,149.085
C06821=1173.406,-7.310,-45.379,179.882,5.884,149.085
C06822=1173.400,-7.061,-45.392,179.884,5.885,149.084
C06823=1173.396,-6.811,-45.405,179.886,5.885,149.083
C06824=1173.390,-6.562,-45.419,179.889,5.886,149.083
C06825=1173.386,-6.312,-45.432,179.891,5.886,149.082
C06826=1173.380,-6.062,-45.445,179.894,5.887,149.082
C06827=1173.376,-5.813,-45.459,179.896,5.887,149.081
C06828=1173.370,-5.563,-45.472,179.899,5.888,149.080
C06829=1173.365,-5.313,-45.485,179.901,5.889,149.080
C06830=1173.360,-5.064,-45.499,179.904,5.889,149.079
C06831=1173.354,-4.815,-45.512,179.906,5.890,149.079
C06832=1173.349,-4.564,-45.525,179.909,5.890,149.078
C06833=1173.344,-4.316,-45.539,179.911,5.891,149.077
C06834=1173.339,-4.065,-45.552,179.914,5.892,149.077
C06835=1173.333,-3.816,-45.565,179.916,5.892,149.076
C06836=1173.329,-3.566,-45.579,179.918,5.893,149.076
C06837=1173.323,-3.317,-45.592,179.921,5.893,149.075
C06838=1173.319,-3.067,-45.606,179.924,5.894,149.074
C06839=1173.313,-2.818,-45.619,179.926,5.895,149.074
C06840=1173.309,-2.568,-45.632,179.929,5.895,149.073
C06841=1173.303,-2.319,-45.646,179.931,5.896,149.072
C06842=1173.299,-2.069,-45.659,179.933,5.896,149.072
C06843=1173.293,-1.820,-45.673,179.936,5.897,149.071
C06844=1173.288,-1.569,-45.686,179.939,5.897,149.071
C06845=1173.283,-1.321,-45.700,179.941,5.898,149.070
C06846=1173.278,-1.070,-45.713,179.944,5.899,149.069
C06847=1173.273,-0.821,-45.727,179.946,5.899,149.069
C06848=1173.268,-0.571,-45.740,179.948,5.900,149.068
C06849=1173.263,-0.321,-45.754,179.951,5.900,149.068
C06850=1173.257,-0.072,-45.767,179.953,5.901,149.067
C06851=1173.253,0.178,-45.781,179.956,5.902,149.066
C06852=1173.247,0.427,-45.795,179.959,5.902,149.066
C06853=1173.242,0.677,-45.808,179.961,5.903,149.065
C06854=1173.237,0.926,-45.821,179.963,5.903,149.065
C06855=1173.232,1.176,-45.836,179.966,5.904,149.064
C06856=1173.226,1.425,-45.848,179.968,5.905,149.063
C06857=1173.222,1.675,-45.863,179.971,5.905,149.063
C06858=1173.216,1.944,-45.878,179.974,5.906,149.062
C06859=1173.211,2.214,-45.893,179.977,5.907,149.061
C06860=1173.205,2.482,-45.907,179.979,5.908,149.061
C06861=1173.200,2.752,-45.921,179.982,5.908,149.060
C06862=1173.195,3.002,-45.935,179.984,5.909,149.060
C06863=1173.189,3.251,-45.949,179.987,5.909,149.059
C06864=1173.185,3.501,-45.962,179.989,5.910,149.058
C06865=1173.179,3.750,-45.976,179.992,5.910,149.058
C06866=1173.174,4.000,-45.990,179.994,5.911,149.057
C06867=1173.169,4.250,-46.004,179.996,5.912,149.057
C06868=1173.164,4.499,-46.017,180.000,5.913,149.056
C06869=1173.159,4.748,-46.031,-179.998,5.914,149.055
C06870=1173.154,4.999,-46.045,-179.995,5.914,149.055
C06871=1173.148,5.248,-46.059,-179.993,5.915,149.054
C06872=1173.144,5.497,-46.072,-179.991,5.916,149.054
C06873=1173.138,5.747,-46.086,-179.988,5.916,149.053
C06874=1173.133,5.996,-46.100,-179.985,5.917,149.052
C06875=1173.128,6.246,-46.114,-179.983,5.917,149.052
C06876=1173.123,6.496,-46.127,-179.980,5.918,149.051
C06877=1173.118,6.745,-46.141,-179.978,5.919,149.051
C06878=1173.113,6.995,-46.155,-179.976,5.919,149.050
C06879=1173.108,7.244,-46.169,-179.973,5.920,149.049
C06880=1173.102,7.494,-46.183,-179.971,5.921,149.049
C06881=1173.098,7.744,-46.197,-179.968,5.921,149.048
C06882=1173.093,7.993,-46.210,-179.966,5.921,149.047
C06883=1173.088,8.242,-46.225,-179.963,5.922,149.047
C06884=1173.083,8.492,-46.239,-179.961,5.923,149.046
C06885=1173.077,8.742,-46.252,-179.958,5.924,149.046
C06886=1173.072,8.991,-46.266,-179.955,5.925,149.045
C06887=1173.068,9.241,-46.280,-179.953,5.925,149.044
C06888=1173.062,9.490,-46.294,-179.950,5.926,149.044
C06889=1173.057,9.740,-46.308,-179.948,5.927,149.043
C06890=1173.052,9.990,-46.322,-179.945,5.927,149.043
C06891=1173.047,10.240,-46.336,-179.943,5.928,149.042
C06892=1173.041,10.489,-46.350,-179.940,5.928,149.041
C06893=1173.036,10.738,-46.364,-179.938,5.929,149.041
C06894=1173.032,10.988,-46.378,-179.936,5.930,149.040
C06895=1173.027,11.237,-46.392,-179.933,5.930,149.040
C06896=1173.022,11.486,-46.406,-179.931,5.931,149.039
C06897=1173.017,11.736,-46.421,-179.928,5.932,149.038
C06898=1173.012,11.986,-46.435,-179.925,5.933,149.038
C06899=1173.006,12.235,-46.448,-179.923,5.934,149.037
C06900=1173.001,12.485,-46.462,-179.920,5.934,149.037
C06901=1172.996,12.735,-46.477,-179.917,5.935,149.036
C06902=1172.991,12.985,-46.491,-179.915,5.935,149.036
C06903=1172.986,13.234,-46.505,-179.913,5.936,149.035
C06904=1172.981,13.483,-46.519,-179.910,5.937,149.034
C06905=1172.976,13.733,-46.533,-179.908,5.937,149.034
C06906=1172.971,13.983,-46.548,-179.905,5.938,149.033
C06907=1172.965,14.232,-46.561,-179.903,5.939,149.033
C06908=1172.960,14.481,-46.576,-179.900,5.939,149.032
C06909=1172.955,14.731,-46.590,-179.897,5.940,149.031
C06910=1172.950,14.981,-46.604,-179.895,5.941,149.031
C06911=1172.945,15.230,-46.618,-179.892,5.942,149.030
C06912=1172.940,15.480,-46.633,-179.890,5.943,149.030
C06913=1172.935,15.729,-46.647,-179.887,5.943,149.029
C06914=1172.930,15.979,-46.661,-179.885,5.943,149.028
C06915=1172.925,16.229,-46.675,-179.883,5.944,149.028
C06916=1172.919,16.478,-46.689,-179.880,5.945,149.027
C06917=1172.914,16.727,-46.704,-179.878,5.946,149.027
C06918=1172.910,16.977,-46.719,-179.875,5.947,149.026
C06919=1172.905,17.226,-46.733,-179.872,5.947,149.025
C06920=1172.900,17.476,-46.747,-179.870,5.948,149.025
C06921=1172.895,17.726,-46.761,-179.867,5.949,149.024
C06922=1172.889,17.975,-46.775,-179.864,5.949,149.023
C06923=1172.884,18.224,-46.790,-179.862,5.950,149.023
C06924=1172.879,18.474,-46.804,-179.860,5.951,149.022
C06925=1172.874,18.724,-46.818,-179.857,5.951,149.022
C06926=1172.870,18.973,-46.833,-179.854,5.953,149.021
C06927=1172.865,19.223,-46.847,-179.852,5.953,149.020
C06928=1172.859,19.472,-46.861,-179.849,5.954,149.020
C06929=1172.854,19.721,-46.876,-179.847,5.954,149.019
C06930=1172.849,19.971,-46.890,-179.845,5.955,149.019
C06931=1172.844,20.221,-46.905,-179.842,5.956,149.018
C06932=1172.839,20.470,-46.920,-179.839,5.956,149.018
C06933=1172.834,20.720,-46.934,-179.837,5.957,149.017
C06934=1172.829,20.970,-46.948,-179.834,5.958,149.016
C06935=1172.824,21.219,-46.963,-179.831,5.959,149.016
C06936=1172.819,21.468,-46.977,-179.829,5.960,149.015
C06937=1172.814,21.717,-46.991,-179.826,5.960,149.015
C06938=1172.808,21.967,-47.006,-179.824,5.961,149.014
C06939=1172.803,22.217,-47.021,-179.822,5.962,149.013
C06940=1172.799,22.466,-47.036,-179.819,5.962,149.013
C06941=1172.794,22.716,-47.050,-179.816,5.964,149.012
C06942=1172.789,22.966,-47.064,-179.814,5.964,149.012
C06943=1172.784,23.215,-47.078,-179.811,5.965,149.011
C06944=1172.778,23.465,-47.094,-179.809,5.965,149.010
C06945=1172.773,23.714,-47.108,-179.806,5.966,149.010
C06946=1172.768,23.964,-47.123,-179.804,5.967,149.009
C06947=1172.763,24.213,-47.137,-179.801,5.968,149.009
C06948=1172.758,24.462,-47.151,-179.799,5.969,149.008
C06949=1172.753,24.712,-47.166,-179.796,5.969,149.008
C06950=1172.748,24.961,-47.181,-179.793,5.970,149.007
C06951=1172.743,25.211,-47.196,-179.791,5.971,149.006
C06952=1172.738,25.460,-47.211,-179.788,5.971,149.006
C06953=1172.733,25.710,-47.225,-179.786,5.973,149.005
C06954=1172.728,25.960,-47.240,-179.783,5.973,149.005
C06955=1172.723,26.209,-47.255,-179.780,5.974,149.004
C06956=1172.718,26.459,-47.269,-179.778,5.975,149.003
C06957=1172.713,26.708,-47.285,-179.776,5.975,149.003
C06958=1172.708,26.958,-47.299,-179.773,5.976,149.002
C06959=1172.703,27.208,-47.313,-179.770,5.977,149.002
C06960=1172.697,27.457,-47.329,-179.768,5.978,149.001
C06961=1172.692,27.707,-47.343,-179.765,5.979,149.001
C06962=1172.687,27.975,-47.359,-179.763,5.979,149.000
C06963=1172.681,28.245,-47.375,-179.759,5.980,148.999
C06964=1172.676,28.513,-47.391,-179.757,5.981,148.999
C06965=1172.671,28.782,-47.406,-179.755,5.982,148.998
C06966=1172.666,29.032,-47.422,-179.751,5.983,148.997
C06967=1172.661,29.281,-47.436,-179.749,5.984,148.997
C06968=1172.656,29.530,-47.451,-179.747,5.984,148.996
C06969=1172.651,29.780,-47.467,-179.744,5.985,148.996
C06970=1172.646,30.029,-47.481,-179.742,5.986,148.995
C06971=1172.640,30.279,-47.497,-179.739,5.986,148.994
C06972=1172.636,30.529,-47.511,-179.736,5.988,148.994
C06973=1172.631,30.778,-47.526,-179.734,5.988,148.993
C06974=1172.625,31.028,-47.541,-179.731,5.989,148.993
C06975=1172.621,31.277,-47.556,-179.729,5.990,148.992
C06976=1172.616,31.527,-47.570,-179.726,5.990,148.992
C06977=1172.610,31.776,-47.586,-179.723,5.992,148.991
C06978=1172.606,32.025,-47.601,-179.721,5.992,148.990
C06979=1172.600,32.275,-47.616,-179.718,5.993,148.990
C06980=1172.595,32.524,-47.631,-179.716,5.994,148.989
C06981=1172.591,32.773,-47.646,-179.714,5.994,148.989
C06982=1172.585,33.023,-47.660,-179.710,5.996,148.988
C06983=1172.581,33.273,-47.676,-179.708,5.996,148.987
C06984=1172.575,33.523,-47.691,-179.705,5.997,148.987
C06985=1172.570,33.772,-47.706,-179.703,5.998,148.986
C06986=1172.565,34.022,-47.721,-179.700,5.999,148.986
C06987=1172.560,34.271,-47.736,-179.698,6.000,148.985
C06988=1172.555,34.521,-47.751,-179.695,6.000,148.985
C06989=1172.550,34.770,-47.766,-179.693,6.001,148.984
C06990=1172.545,35.019,-47.782,-179.690,6.002,148.983
C06991=1172.540,35.269,-47.796,-179.687,6.003,148.983
C06992=1172.534,35.518,-47.812,-179.685,6.004,148.982
C06993=1172.530,35.768,-47.827,-179.682,6.004,148.982
C06994=1172.525,36.017,-47.843,-179.680,6.005,148.981
C06995=1172.520,36.267,-47.857,-179.677,6.007,148.980
C06996=1172.515,36.517,-47.872,-179.674,6.007,148.980
C06997=1172.510,36.766,-47.887,-179.672,6.008,148.979
C06998=1172.505,37.015,-47.903,-179.670,6.008,148.979
C06999=1172.500,37.265,-47.917,-179.667,6.009,148.978
C07000=1172.494,37.514,-47.933,-179.664,6.011,148.978
C07001=1172.490,37.764,-47.948,-179.662,6.011,148.977
C07002=1172.485,38.013,-47.964,-179.659,6.012,148.976
C07003=1172.480,38.262,-47.979,-179.657,6.012,148.976
C07004=1172.475,38.512,-47.994,-179.654,6.014,148.975
C07005=1172.469,38.762,-48.009,-179.651,6.015,148.975
C07006=1172.464,39.011,-48.024,-179.649,6.015,148.974
C07007=1172.460,39.261,-48.040,-179.647,6.016,148.974
C07008=1172.455,39.510,-48.055,-179.643,6.017,148.973
C07009=1172.450,39.760,-48.071,-179.641,6.018,148.972
C07010=1172.444,40.009,-48.086,-179.639,6.019,148.972
C07011=1172.440,40.258,-48.101,-179.636,6.019,148.971
C07012=1172.435,40.508,-48.117,-179.633,6.021,148.971
C07013=1172.430,40.757,-48.132,-179.631,6.022,148.970
C07014=1172.424,41.007,-48.147,-179.628,6.022,148.970
C07015=1172.419,41.257,-48.163,-179.626,6.023,148.969
C07016=1172.414,41.506,-48.178,-179.623,6.024,148.968
C07017=1172.410,41.756,-48.194,-179.620,6.025,148.968
C07018=1172.404,42.005,-48.209,-179.618,6.026,148.967
C07019=1172.400,42.254,-48.224,-179.616,6.026,148.967
C07020=1172.394,42.504,-48.240,-179.613,6.028,148.966
C07021=1172.389,42.753,-48.255,-179.610,6.028,148.965
C07022=1172.385,43.003,-48.271,-179.608,6.029,148.965
C07023=1172.379,43.252,-48.286,-179.605,6.030,148.964
C07024=1172.374,43.502,-48.302,-179.602,6.031,148.964
C07025=1172.369,43.751,-48.317,-179.600,6.032,148.963
C07026=1172.365,44.001,-48.333,-179.597,6.032,148.963
C07027=1172.359,44.250,-48.349,-179.595,6.034,148.962
C07028=1172.355,44.499,-48.364,-179.592,6.034,148.961
C07029=1172.349,44.749,-48.379,-179.590,6.035,148.961
C07030=1172.345,44.998,-48.396,-179.587,6.036,148.960
C07031=1172.339,45.248,-48.411,-179.584,6.037,148.960
C07032=1172.335,45.497,-48.426,-179.582,6.038,148.959
C07033=1172.330,45.747,-48.442,-179.579,6.038,148.959
C07034=1172.324,45.996,-48.458,-179.576,6.040,148.958
C07035=1172.319,46.246,-48.473,-179.574,6.041,148.957
C07036=1172.315,46.496,-48.489,-179.572,6.042,148.957
C07037=1172.310,46.745,-48.504,-179.569,6.042,148.956
C07038=1172.304,46.994,-48.520,-179.566,6.044,148.956
C07039=1172.299,47.243,-48.536,-179.564,6.044,148.955
C07040=1172.294,47.493,-48.552,-179.561,6.045,148.955
C07041=1172.290,47.742,-48.567,-179.558,6.046,148.954
C07042=1172.284,47.992,-48.583,-179.556,6.047,148.953
C07043=1172.280,48.242,-48.599,-179.553,6.048,148.953
C07044=1172.274,48.491,-48.615,-179.550,6.049,148.952
C07045=1172.269,48.740,-48.631,-179.548,6.050,148.952
C07046=1172.265,48.990,-48.646,-179.545,6.050,148.951
C07047=1172.260,49.239,-48.662,-179.543,6.051,148.951
C07048=1172.254,49.489,-48.677,-179.540,6.053,148.950
C07049=1172.250,49.738,-48.694,-179.538,6.053,148.950
C07050=1172.244,49.987,-48.710,-179.535,6.054,148.949
C07051=1172.240,50.238,-48.725,-179.532,6.056,148.949
C07052=1172.235,50.486,-48.742,-179.530,6.056,148.948
C07053=1172.230,50.735,-48.757,-179.527,6.057,148.947
C07054=1172.225,50.986,-48.773,-179.524,6.058,148.947
C07055=1172.220,51.235,-48.788,-179.522,6.059,148.946
C07056=1172.215,51.484,-48.805,-179.520,6.060,148.946
C07057=1172.210,51.734,-48.821,-179.516,6.061,148.945
C07058=1172.204,51.983,-48.836,-179.514,6.062,148.945
C07059=1172.200,52.233,-48.853,-179.512,6.062,148.944
C07060=1172.195,52.482,-48.868,-179.509,6.064,148.943
C07061=1172.189,52.732,-48.884,-179.506,6.065,148.943
C07062=1172.185,52.981,-48.901,-179.504,6.065,148.942
C07063=1172.180,53.230,-48.916,-179.501,6.067,148.942
C07064=1172.176,53.480,-48.932,-179.499,6.068,148.941
C07065=1172.170,53.729,-48.948,-179.496,6.068,148.941
C07066=1172.165,53.997,-48.965,-179.493,6.069,148.940
C07067=1172.160,54.267,-48.982,-179.491,6.070,148.939
C07068=1172.154,54.535,-48.999,-179.487,6.072,148.939
C07069=1172.148,54.803,-49.018,-179.485,6.072,148.938
C07070=1172.144,55.053,-49.033,-179.482,6.074,148.938
C07071=1172.139,55.302,-49.049,-179.479,6.074,148.937
C07072=1172.133,55.552,-49.065,-179.477,6.075,148.937
C07073=1172.128,55.802,-49.081,-179.474,6.077,148.936
C07074=1172.123,56.050,-49.098,-179.472,6.077,148.936
C07075=1172.118,56.301,-49.114,-179.469,6.078,148.935
C07076=1172.113,56.549,-49.130,-179.466,6.079,148.934
C07077=1172.108,56.799,-49.146,-179.464,6.080,148.934
C07078=1172.103,57.048,-49.162,-179.461,6.081,148.933
C07079=1172.098,57.298,-49.178,-179.459,6.082,148.933
C07080=1172.093,57.547,-49.195,-179.456,6.083,148.932
C07081=1172.089,57.797,-49.211,-179.453,6.084,148.932
C07082=1172.084,58.046,-49.227,-179.451,6.085,148.931
C07083=1172.079,58.296,-49.243,-179.448,6.086,148.930
C07084=1172.074,58.545,-49.259,-179.445,6.087,148.930
C07085=1172.069,58.794,-49.276,-179.443,6.088,148.929
C07086=1172.064,59.044,-49.291,-179.440,6.089,148.929
C07087=1172.059,59.293,-49.308,-179.438,6.090,148.928
C07088=1172.054,59.542,-49.324,-179.435,6.091,148.928
C07089=1172.049,59.793,-49.341,-179.432,6.092,148.927
C07090=1172.044,60.041,-49.357,-179.430,6.093,148.926
C07091=1172.039,60.291,-49.374,-179.428,6.094,148.926
C07092=1172.034,60.540,-49.389,-179.424,6.095,148.925
C07093=1172.029,60.790,-49.406,-179.422,6.096,148.925
C07094=1172.024,61.038,-49.422,-179.420,6.097,148.924
C07095=1172.019,61.289,-49.438,-179.417,6.098,148.924
C07096=1172.014,61.538,-49.455,-179.414,6.099,148.923
C07097=1172.009,61.787,-49.472,-179.411,6.100,148.923
C07098=1172.004,62.037,-49.488,-179.409,6.101,148.922
C07099=1171.999,62.286,-49.504,-179.407,6.102,148.922
C07100=1171.995,62.535,-49.521,-179.403,6.103,148.921
C07101=1171.989,62.785,-49.536,-179.401,6.104,148.921
C07102=1171.984,63.035,-49.554,-179.398,6.105,148.920
C07103=1171.979,63.283,-49.570,-179.396,6.106,148.919
C07104=1171.975,63.533,-49.587,-179.393,6.107,148.919
C07105=1171.970,63.783,-49.603,-179.391,6.108,148.918
C07106=1171.965,64.032,-49.619,-179.388,6.109,148.918
C07107=1171.960,64.282,-49.636,-179.385,6.111,148.917
C07108=1171.954,64.530,-49.652,-179.383,6.111,148.917
C07109=1171.950,64.780,-49.669,-179.380,6.112,148.916
C07110=1171.945,65.030,-49.685,-179.377,6.113,148.915
C07111=1171.939,65.279,-49.702,-179.375,6.114,148.915
C07112=1171.935,65.529,-49.719,-179.372,6.116,148.914
C07113=1171.930,65.778,-49.735,-179.370,6.116,148.914
C07114=1171.925,66.027,-49.752,-179.367,6.117,148.913
C07115=1171.920,66.277,-49.769,-179.364,6.119,148.913
C07116=1171.916,66.526,-49.786,-179.362,6.119,148.912
C07117=1171.910,66.776,-49.801,-179.359,6.121,148.912
C07118=1171.905,67.025,-49.818,-179.356,6.121,148.911
C07119=1171.900,67.274,-49.835,-179.354,6.122,148.911
C07120=1171.895,67.524,-49.851,-179.351,6.124,148.910
C07121=1171.891,67.773,-49.868,-179.349,6.124,148.910
C07122=1171.885,68.022,-49.885,-179.346,6.126,148.909
C07123=1171.881,68.272,-49.902,-179.343,6.127,148.908
C07124=1171.876,68.521,-49.918,-179.341,6.128,148.908
C07125=1171.870,68.770,-49.935,-179.338,6.129,148.907
C07126=1171.866,69.020,-49.952,-179.336,6.130,148.907
C07127=1171.861,69.269,-49.969,-179.333,6.131,148.906
C07128=1171.856,69.519,-49.986,-179.331,6.132,148.906
C07129=1171.851,69.768,-50.002,-179.327,6.133,148.905
C07130=1171.846,70.018,-50.019,-179.325,6.134,148.905
C07131=1171.841,70.267,-50.036,-179.322,6.135,148.904
C07132=1171.836,70.516,-50.052,-179.320,6.136,148.904
C07133=1171.831,70.766,-50.070,-179.317,6.138,148.903
C07134=1171.827,71.015,-50.086,-179.314,6.139,148.903
C07135=1171.821,71.265,-50.104,-179.312,6.139,148.902
C07136=1171.816,71.514,-50.120,-179.309,6.141,148.902
C07137=1171.812,71.763,-50.136,-179.306,6.141,148.901
C07138=1171.807,72.013,-50.154,-179.304,6.143,148.900
C07139=1171.802,72.262,-50.170,-179.301,6.143,148.900
C07140=1171.796,72.512,-50.187,-179.298,6.145,148.899
C07141=1171.792,72.760,-50.205,-179.296,6.146,148.899
C07142=1171.787,73.010,-50.222,-179.293,6.147,148.898
C07143=1171.782,73.259,-50.238,-179.291,6.148,148.898
C07144=1171.777,73.509,-50.256,-179.288,6.149,148.897
C07145=1171.772,73.758,-50.272,-179.285,6.150,148.897
C07146=1171.767,74.008,-50.289,-179.283,6.151,148.896
C07147=1171.762,74.258,-50.306,-179.280,6.153,148.896
C07148=1171.757,74.506,-50.324,-179.277,6.153,148.895
C07149=1171.752,74.756,-50.340,-179.275,6.155,148.895
C07150=1171.747,75.005,-50.358,-179.272,6.155,148.894
C07151=1171.743,75.255,-50.374,-179.269,6.157,148.894
C07152=1171.737,75.504,-50.391,-179.267,6.158,148.893
C07153=1171.733,75.753,-50.409,-179.264,6.159,148.892
C07154=1171.728,76.003,-50.426,-179.262,6.160,148.892
C07155=1171.723,76.252,-50.443,-179.259,6.162,148.891
C07156=1171.718,76.502,-50.460,-179.257,6.162,148.891
C07157=1171.713,76.750,-50.477,-179.253,6.164,148.890
C07158=1171.708,77.000,-50.494,-179.251,6.165,148.890
C07159=1171.703,77.249,-50.511,-179.248,6.166,148.889
C07160=1171.698,77.498,-50.529,-179.246,6.167,148.889
C07161=1171.693,77.748,-50.546,-179.243,6.169,148.888
C07162=1171.689,77.998,-50.563,-179.240,6.169,148.888
C07163=1171.683,78.246,-50.580,-179.238,6.171,148.887
C07164=1171.679,78.496,-50.597,-179.235,6.171,148.887
C07165=1171.674,78.745,-50.614,-179.232,6.173,148.886
C07166=1171.669,78.995,-50.632,-179.230,6.174,148.885
C07167=1171.664,79.244,-50.649,-179.227,6.175,148.885
C07168=1171.659,79.494,-50.666,-179.224,6.176,148.884
C07169=1171.654,79.743,-50.684,-179.222,6.177,148.884
C07170=1171.649,80.011,-50.702,-179.219,6.178,148.883
C07171=1171.643,80.280,-50.721,-179.216,6.180,148.883
C07172=1171.638,80.548,-50.740,-179.213,6.181,148.882
C07173=1171.632,80.816,-50.758,-179.211,6.182,148.882
C07174=1171.628,81.066,-50.775,-179.208,6.183,148.881
C07175=1171.623,81.315,-50.793,-179.206,6.184,148.881
C07176=1171.618,81.565,-50.810,-179.202,6.186,148.880
C07177=1171.614,81.814,-50.828,-179.200,6.186,148.880
C07178=1171.608,82.063,-50.845,-179.197,6.188,148.879
C07179=1171.603,82.313,-50.863,-179.195,6.189,148.879
C07180=1171.599,82.562,-50.880,-179.192,6.190,148.878
C07181=1171.594,82.811,-50.897,-179.190,6.191,148.878
C07182=1171.589,83.061,-50.915,-179.187,6.193,148.877
C07183=1171.584,83.310,-50.933,-179.184,6.194,148.876
C07184=1171.579,83.559,-50.949,-179.181,6.195,148.876
C07185=1171.574,83.808,-50.967,-179.179,6.196,148.876
C07186=1171.569,84.058,-50.984,-179.176,6.197,148.875
C07187=1171.564,84.307,-51.002,-179.173,6.199,148.875
C07188=1171.559,84.557,-51.019,-179.171,6.199,148.874
C07189=1171.554,84.806,-51.037,-179.168,6.201,148.873
C07190=1171.549,85.055,-51.055,-179.165,6.201,148.873
C07191=1171.544,85.305,-51.072,-179.163,6.203,148.872
C07192=1171.539,85.554,-51.090,-179.161,6.204,148.872
C07193=1171.535,85.803,-51.107,-179.157,6.205,148.871
C07194=1171.530,86.053,-51.125,-179.155,6.206,148.871
C07195=1171.525,86.302,-51.143,-179.152,6.208,148.870
C07196=1171.520,86.552,-51.160,-179.150,6.209,148.870
C07197=1171.515,86.801,-51.178,-179.147,6.210,148.869
C07198=1171.511,87.050,-51.195,-179.144,6.212,148.869
C07199=1171.506,87.299,-51.213,-179.142,6.212,148.868
C07200=1171.501,87.549,-51.231,-179.139,6.214,148.868
C07201=1171.496,87.798,-51.249,-179.136,6.215,148.867
C07202=1171.490,88.048,-51.266,-179.134,6.216,148.867
C07203=1171.486,88.297,-51.284,-179.131,6.217,148.866
C07204=1171.481,88.546,-51.302,-179.128,6.219,148.866
C07205=1171.476,88.795,-51.320,-179.126,6.220,148.865
C07206=1171.471,89.045,-51.336,-179.123,6.221,148.865
C07207=1171.466,89.294,-51.354,-179.120,6.223,148.864
C07208=1171.461,89.543,-51.372,-179.118,6.223,148.864
C07209=1171.457,89.792,-51.390,-179.115,6.225,148.863
C07210=1171.451,90.042,-51.408,-179.113,6.226,148.863
C07211=1171.446,90.291,-51.426,-179.110,6.227,148.862
C07212=1171.442,90.541,-51.444,-179.107,6.228,148.862
C07213=1171.437,90.790,-51.462,-179.104,6.229,148.861
C07214=1171.432,91.039,-51.480,-179.102,6.231,148.861
C07215=1171.427,91.288,-51.498,-179.099,6.232,148.860
C07216=1171.422,91.538,-51.515,-179.096,6.233,148.860
C07217=1171.417,91.787,-51.533,-179.094,6.234,148.859
C07218=1171.412,92.037,-51.551,-179.091,6.236,148.859
C07219=1171.407,92.286,-51.569,-179.089,6.236,148.858
C07220=1171.402,92.535,-51.587,-179.086,6.238,148.858
C07221=1171.398,92.784,-51.605,-179.083,6.239,148.857
C07222=1171.393,93.033,-51.623,-179.081,6.240,148.857
C07223=1171.388,93.282,-51.641,-179.078,6.242,148.856
C07224=1171.383,93.532,-51.659,-179.075,6.243,148.856
C07225=1171.379,93.782,-51.677,-179.073,6.244,148.855
C07226=1171.373,94.031,-51.695,-179.070,6.246,148.855
C07227=1171.368,94.280,-51.713,-179.067,6.247,148.854
C07228=1171.363,94.530,-51.731,-179.065,6.248,148.854
C07229=1171.359,94.779,-51.749,-179.062,6.249,148.853
C07230=1171.354,95.028,-51.767,-179.059,6.251,148.853
C07231=1171.349,95.278,-51.785,-179.056,6.252,148.852
C07232=1171.344,95.527,-51.803,-179.054,6.253,148.852
C07233=1171.340,95.776,-51.821,-179.051,6.255,148.851
C07234=1171.335,96.025,-51.839,-179.049,6.255,148.851
C07235=1171.330,96.275,-51.857,-179.046,6.257,148.850
C07236=1171.325,96.524,-51.875,-179.043,6.258,148.850
C07237=1171.320,96.772,-51.894,-179.041,6.259,148.849
C07238=1171.315,97.023,-51.912,-179.038,6.261,148.849
C07239=1171.310,97.272,-51.930,-179.035,6.262,148.848
C07240=1171.305,97.521,-51.948,-179.033,6.263,148.848
C07241=1171.300,97.770,-51.966,-179.030,6.265,148.847
C07242=1171.295,98.019,-51.984,-179.028,6.266,148.847
C07243=1171.291,98.269,-52.003,-179.025,6.267,148.846
C07244=1171.286,98.518,-52.021,-179.022,6.269,148.846
C07245=1171.281,98.768,-52.039,-179.019,6.270,148.845
C07246=1171.276,99.016,-52.058,-179.016,6.271,148.845
C07247=1171.271,99.265,-52.076,-179.014,6.273,148.844
C07248=1171.267,99.515,-52.094,-179.011,6.274,148.844
C07249=1171.262,99.765,-52.112,-179.008,6.275,148.843
C07250=1171.257,100.014,-52.130,-179.006,6.276,148.843
C07251=1171.251,100.263,-52.149,-179.003,6.277,148.842
C07252=1171.247,100.512,-52.168,-179.000,6.279,148.842
C07253=1171.242,100.762,-52.186,-178.998,6.280,148.841
C07254=1171.237,101.011,-52.204,-178.995,6.281,148.841
C07255=1171.232,101.260,-52.222,-178.992,6.283,148.840
C07256=1171.228,101.510,-52.242,-178.990,6.284,148.840
C07257=1171.223,101.759,-52.259,-178.987,6.285,148.839
C07258=1171.218,102.008,-52.277,-178.985,6.287,148.839
C07259=1171.212,102.257,-52.296,-178.982,6.288,148.838
C07260=1171.208,102.507,-52.315,-178.979,6.289,148.838
C07261=1171.203,102.756,-52.333,-178.976,6.291,148.837
C07262=1171.199,103.005,-52.351,-178.974,6.292,148.837
C07263=1171.194,103.255,-52.371,-178.971,6.293,148.836
C07264=1171.189,103.504,-52.389,-178.968,6.295,148.836
C07265=1171.184,103.753,-52.407,-178.966,6.296,148.835
C07266=1171.179,104.002,-52.426,-178.963,6.297,148.835
C07267=1171.174,104.252,-52.444,-178.961,6.298,148.835
C07268=1171.169,104.501,-52.462,-178.958,6.300,148.834
C07269=1171.165,104.749,-52.481,-178.955,6.301,148.834
C07270=1171.160,105.000,-52.500,-178.952,6.303,148.833
C07271=1171.155,105.248,-52.519,-178.950,6.304,148.832
C07272=1171.149,105.498,-52.537,-178.947,6.305,148.832
C07273=1171.145,105.748,-52.556,-178.944,6.307,148.832
C07274=1171.140,106.015,-52.576,-178.942,6.308,148.831
C07275=1171.135,106.284,-52.596,-178.939,6.309,148.831
C07276=1171.129,106.552,-52.615,-178.936,6.311,148.830
C07277=1171.125,106.821,-52.636,-178.933,6.312,148.830
C07278=1171.120,107.070,-52.654,-178.930,6.314,148.829
C07279=1171.114,107.319,-52.673,-178.928,6.315,148.828
C07280=1171.110,107.569,-52.692,-178.925,6.316,148.828
C07281=1171.105,107.817,-52.711,-178.922,6.318,148.828
C07282=1171.100,108.067,-52.729,-178.920,6.319,148.827
C07283=1171.096,108.316,-52.748,-178.917,6.320,148.827
C07284=1171.090,108.565,-52.767,-178.914,6.322,148.826
C07285=1171.086,108.815,-52.786,-178.911,6.323,148.826
C07286=1171.080,109.064,-52.804,-178.909,6.324,148.825
C07287=1171.076,109.313,-52.823,-178.906,6.326,148.825
C07288=1171.071,109.562,-52.843,-178.903,6.328,148.824
C07289=1171.066,109.811,-52.861,-178.901,6.328,148.824
C07290=1171.061,110.061,-52.880,-178.898,6.330,148.823
C07291=1171.057,110.310,-52.898,-178.895,6.332,148.823
C07292=1171.052,110.560,-52.918,-178.893,6.332,148.822
C07293=1171.047,110.808,-52.937,-178.890,6.334,148.822
C07294=1171.042,111.058,-52.955,-178.887,6.336,148.821
C07295=1171.038,111.307,-52.974,-178.885,6.337,148.821
C07296=1171.032,111.556,-52.994,-178.882,6.338,148.820
C07297=1171.028,111.806,-53.012,-178.879,6.340,148.820
C07298=1171.023,112.055,-53.031,-178.877,6.341,148.820
C07299=1171.019,112.304,-53.050,-178.874,6.343,148.819
C07300=1171.013,112.553,-53.069,-178.871,6.344,148.819
C07301=1171.009,112.803,-53.088,-178.869,6.345,148.818
C07302=1171.004,113.051,-53.107,-178.866,6.347,148.818
C07303=1170.998,113.302,-53.126,-178.863,6.348,148.817
C07304=1170.994,113.550,-53.145,-178.861,6.349,148.817
C07305=1170.989,113.799,-53.164,-178.858,6.351,148.816
C07306=1170.985,114.048,-53.183,-178.855,6.353,148.816
C07307=1170.979,114.297,-53.202,-178.853,6.353,148.815
C07308=1170.974,114.547,-53.221,-178.850,6.355,148.815
C07309=1170.970,114.796,-53.240,-178.847,6.357,148.814
C07310=1170.965,115.046,-53.260,-178.844,6.359,148.814
C07311=1170.960,115.294,-53.278,-178.842,6.359,148.813
C07312=1170.955,115.544,-53.298,-178.839,6.361,148.813
C07313=1170.950,115.793,-53.317,-178.836,6.363,148.813
C07314=1170.946,116.042,-53.336,-178.834,6.364,148.812
C07315=1170.941,116.292,-53.355,-178.831,6.365,148.812
C07316=1170.936,116.541,-53.375,-178.828,6.367,148.811
C07317=1170.932,116.790,-53.394,-178.826,6.368,148.811
C07318=1170.926,117.039,-53.413,-178.823,6.370,148.810
C07319=1170.922,117.289,-53.433,-178.820,6.371,148.810
C07320=1170.917,117.537,-53.451,-178.818,6.372,148.809
C07321=1170.912,117.787,-53.470,-178.815,6.374,148.809
C07322=1170.907,118.036,-53.490,-178.812,6.376,148.809
C07323=1170.902,118.286,-53.509,-178.810,6.376,148.808
C07324=1170.897,118.534,-53.528,-178.807,6.378,148.808
C07325=1170.893,118.784,-53.548,-178.804,6.380,148.807
C07326=1170.888,119.033,-53.567,-178.801,6.382,148.807
C07327=1170.883,119.282,-53.586,-178.799,6.382,148.806
